# B&R Automation Studio project OpcUaSample410_BrbLibUa103 (part 7)

#### BrbUint64FromString.c
```c
#include <bur/plctypes.h>
#ifdef __cplusplus
	extern "C"
	{
#endif

#include "BrbLib.h"
#include <string.h>

#ifdef __cplusplus
	};
#endif

// NOLINTBEGIN(readability-*, bugprone-easily-swappable-parameters, clang-diagnostic-invalid-utf8, clang-diagnostic-invalid-source-encoding, clang-diagnostic-pointer-arith, clang-diagnostic-strict-prototypes, hicpp-uppercase-literal-suffix, cppcoreguidelines-*, performance-*)

// Die Matrix enthält für alle Dezimal-Wertigkeiten (0..9) jeder Stelle (0..19) die Bit-Wertigkeiten für Low+High
const BrbUint64_TYP BRBR_UINT64_FROMSTRING_MATRIX[20][10] =
	{
	//																0	Low      , High					1	Low      , High					2	Low      , High					3	Low      , High					4	Low      , High					5	Low      , High					6	Low      , High					7	Low      , High					8	Low      , High					9	Low      , High
	/* 00 = 1  */										{	{0x00000000, 0x00000000}, {0x00000001, 0x00000000}, {0x00000002, 0x00000000}, {0x00000003, 0x00000000}, {0x00000004, 0x00000000}, {0x00000005, 0x00000000}, {0x00000006, 0x00000000}, {0x00000007, 0x00000000}, {0x00000008, 0x00000000}, {0x00000009, 0x00000000}},
	/* 01 = 10 */										{	{0x00000000, 0x00000000}, {0x0000000A, 0x00000000}, {0x00000014, 0x00000000}, {0x0000001E, 0x00000000}, {0x00000028, 0x00000000}, {0x00000032, 0x00000000}, {0x0000003C, 0x00000000}, {0x00000046, 0x00000000}, {0x00000050, 0x00000000}, {0x0000005A, 0x00000000}},
	/* 02 = 100 */									{	{0x00000000, 0x00000000}, {0x00000064, 0x00000000}, {0x000000C8, 0x00000000}, {0x0000012C, 0x00000000}, {0x00000190, 0x00000000}, {0x000001F4, 0x00000000}, {0x00000258, 0x00000000}, {0x000002BC, 0x00000000}, {0x00000320, 0x00000000}, {0x00000384, 0x00000000}},
	/* 03 = 1000 */									{	{0x00000000, 0x00000000}, {0x000003E8, 0x00000000}, {0x000007D0, 0x00000000}, {0x00000BB8, 0x00000000}, {0x00000FA0, 0x00000000}, {0x00001388, 0x00000000}, {0x00001770, 0x00000000}, {0x00001B58, 0x00000000}, {0x00001F40, 0x00000000}, {0x00002328, 0x00000000}},
	/* 04 = 10000 */								{	{0x00000000, 0x00000000}, {0x00002710, 0x00000000}, {0x00004E20, 0x00000000}, {0x00007530, 0x00000000}, {0x00009C40, 0x00000000}, {0x0000C350, 0x00000000}, {0x0000EA60, 0x00000000}, {0x00011170, 0x00000000}, {0x00013880, 0x00000000}, {0x00015F90, 0x00000000}},
	/* 05 = 100000 */								{	{0x00000000, 0x00000000}, {0x000186A0, 0x00000000}, {0x00030D40, 0x00000000}, {0x000493E0, 0x00000000}, {0x00061A80, 0x00000000}, {0x0007A120, 0x00000000}, {0x000927C0, 0x00000000}, {0x000AAE60, 0x00000000}, {0x000C3500, 0x00000000}, {0x000DBBA0, 0x00000000}},
	/* 06 = 1000000 */							{	{0x00000000, 0x00000000}, {0x000F4240, 0x00000000}, {0x001E8480, 0x00000000}, {0x002DC6C0, 0x00000000}, {0x003D0900, 0x00000000}, {0x004C4B40, 0x00000000}, {0x005B8D80, 0x00000000}, {0x006ACFC0, 0x00000000}, {0x007A1200, 0x00000000}, {0x00895440, 0x00000000}},
	/* 07 = 10000000 */							{	{0x00000000, 0x00000000}, {0x00989680, 0x00000000}, {0x01312D00, 0x00000000}, {0x01C9C380, 0x00000000}, {0x02625A00, 0x00000000}, {0x02FAF080, 0x00000000}, {0x03938700, 0x00000000}, {0x042C1D80, 0x00000000}, {0x04C4B400, 0x00000000}, {0x055D4A80, 0x00000000}},
	/* 08 = 100000000 */						{	{0x00000000, 0x00000000}, {0x05F5E100, 0x00000000}, {0x0BEBC200, 0x00000000}, {0x11E1A300, 0x00000000}, {0x17D78400, 0x00000000}, {0x1DCD6500, 0x00000000}, {0x23C34600, 0x00000000}, {0x29B92700, 0x00000000}, {0x2FAF0800, 0x00000000}, {0x35A4E900, 0x00000000}},
	/* 09 = 1000000000 */						{	{0x00000000, 0x00000000}, {0x3B9ACA00, 0x00000000}, {0x77359400, 0x00000000}, {0xB2D05E00, 0x00000000}, {0xEE6B2800, 0x00000000}, {0x2A05F200, 0x00000001}, {0x65A0BC00, 0x00000001}, {0xA13B8600, 0x00000001}, {0xDCD65000, 0x00000001}, {0x18711A00, 0x00000002}},
	/* 10 = 10000000000 */					{	{0x00000000, 0x00000000}, {0x540BE400, 0x00000002}, {0xA817C800, 0x00000004}, {0xFC23AC00, 0x00000006}, {0x502F9000, 0x00000009}, {0xA43B7400, 0x0000000B}, {0xF8475800, 0x0000000D}, {0x4C533C00, 0x00000010}, {0xA05F2000, 0x00000012}, {0xF46B0400, 0x00000014}},
	/* 11 = 100000000000 */					{	{0x00000000, 0x00000000}, {0x4876E800, 0x00000017}, {0x90EDD000, 0x0000002E}, {0xD964B800, 0x00000045}, {0x21DBA000, 0x0000005D}, {0x6A528800, 0x00000074}, {0xB2C97000, 0x0000008B}, {0xFB405800, 0x000000A2}, {0x43B74000, 0x000000BA}, {0x8C2E2800, 0x000000D1}},
	/* 12 = 1000000000000 */				{	{0x00000000, 0x00000000}, {0xD4A51000, 0x000000E8}, {0xA94A2000, 0x000001D1}, {0x7DEF3000, 0x000002BA}, {0x52944000, 0x000003A3}, {0x27395000, 0x0000048C}, {0xFBDE6000, 0x00000574}, {0xD0837000, 0x0000065D}, {0xA5288000, 0x00000746}, {0x79CD9000, 0x0000082F}},
	/* 13 = 10000000000000 */				{	{0x00000000, 0x00000000}, {0x4E72A000, 0x00000918}, {0x9CE54000, 0x00001230}, {0xEB57E000, 0x00001B48}, {0x39CA8000, 0x00002461}, {0x883D2000, 0x00002D79}, {0xD6AFC000, 0x00003691}, {0x25226000, 0x00003FAA}, {0x73950000, 0x000048C2}, {0xC207A000, 0x000051DA}},
	/* 14 = 100000000000000 */			{	{0x00000000, 0x00000000}, {0x107A4000, 0x00005AF3}, {0x20F48000, 0x0000B5E6}, {0x316EC000, 0x000110D9}, {0x41E90000, 0x00016BCC}, {0x52634000, 0x0001C6BF}, {0x62DD8000, 0x000221B2}, {0x7357C000, 0x00027CA5}, {0x83D20000, 0x0002D798}, {0x944C4000, 0x0003328B}},
	/* 15 = 1000000000000000 */			{	{0x00000000, 0x00000000}, {0xA4C68000, 0x00038D7E}, {0x498D0000, 0x00071AFD}, {0xEE538000, 0x000AA87B}, {0x931A0000, 0x000E35FA}, {0x37E08000, 0x0011C379}, {0xDCA70000, 0x001550F7}, {0x816D8000, 0x0018DE76}, {0x26340000, 0x001C6BF5}, {0xCAFA8000, 0x001FF973}},
	/* 16 = 10000000000000000 */		{	{0x00000000, 0x00000000}, {0x6FC10000, 0x002386F2}, {0xDF820000, 0x00470DE4}, {0x4F430000, 0x006A94D7}, {0xBF040000, 0x008E1BC9}, {0x2EC50000, 0x00B1A2BC}, {0x9E860000, 0x00D529AE}, {0x0E470000, 0x00F8B0A1}, {0x7E080000, 0x011C3793}, {0xEDC90000, 0x013FBE85}},
	/* 17 = 100000000000000000 */		{	{0x00000000, 0x00000000}, {0x5D8A0000, 0x01634578}, {0xBB140000, 0x02C68AF0}, {0x189E0000, 0x0429D069}, {0x76280000, 0x058D15E1}, {0xD3B20000, 0x06F05B59}, {0x313C0000, 0x0853A0D2}, {0x8EC60000, 0x09B6E64A}, {0xEC500000, 0x0B1A2BC2}, {0x49DA0000, 0x0C7D713B}},
	/* 18 = 1000000000000000000 */	{	{0x00000000, 0x00000000}, {0xA7640000, 0x0DE0B6B3}, {0x4EC80000, 0x1BC16D67}, {0xF62C0000, 0x29A2241A}, {0x9D900000, 0x3782DACE}, {0x44F40000, 0x45639182}, {0xEC580000, 0x53444835}, {0x93BC0000, 0x6124FEE9}, {0x3B200000, 0x6F05B59D}, {0xE2840000, 0x7CE66C50}},
	/* 19 = 10000000000000000000 */	{	{0x00000000, 0x00000000}, {0x89E80000, 0x8AC72304}, {0x00000000, 0x00000000}, {0x00000000, 0x00000000}, {0x00000000, 0x00000000}, {0x00000000, 0x00000000}, {0x00000000, 0x00000000}, {0x00000000, 0x00000000}, {0x00000000, 0x00000000}, {0x00000000, 0x00000000}},
	};

/* Wandelt einen Uint64-Wert zu einem String */
signed long BrbUint64FromString(struct BrbUint64_TYP* pUint64, plcstring* pText)
{
	if(pUint64 == 0 || pText == 0)
	{
		return eBRB_ERR_NULL_POINTER;
	}
	pUint64->nLow = 0;
	pUint64->nHigh = 0;
	UDINT nTextLen = strlen(pText);
	if(nTextLen >= nBRB_UINT64_CHAR_MAX)
	{
		return eBRB_ERR_STRING_TOO_LONG;
	}
	DINT eResult = eBRB_ERR_OK;
	UDINT nDigit = 0; // Stelle von hinten
	STRING* pChar = 0;
	USINT nDigitVal = 0; // Wert der Stelle als Einer-Wertigkeit
	const BrbUint64_TYP* pOperand = 0; // Zeiger auf die Wertigkeits-Matrix
	for(nDigit=0; nDigit<nTextLen; nDigit++)
	{
		pChar = (STRING*)pText+(nTextLen-1-nDigit);
		if(*pChar >= '0' && *pChar <= '9')
		{
			// Zeichen ist eine Nummer
			nDigitVal = (USINT)(*pChar-'0'); // Wert als Einer-Stelle
			pOperand = &BRBR_UINT64_FROMSTRING_MATRIX[nDigit][nDigitVal];
			DINT nStatus = BrbByteArrayAdd((USINT*)pUint64, 8, (USINT*)pOperand, 8);
			if(nStatus != eBRB_ERR_OK)
			{
				// Überlauf -> Abbrechen
				eResult = nStatus;
				break;
			}
		}
		else
		{
			// Zeichen ist keine Nummer -> Abbrechen
			break;
		}
	}
	return eResult;
}

// NOLINTEND(readability-*, bugprone-easily-swappable-parameters, clang-diagnostic-invalid-utf8, clang-diagnostic-invalid-source-encoding, clang-diagnostic-pointer-arith, clang-diagnostic-strict-prototypes, hicpp-uppercase-literal-suffix, cppcoreguidelines-*, performance-*)
```

#### BrbUint64ToString.c
```c
#include <bur/plctypes.h>
#ifdef __cplusplus
	extern "C"
	{
#endif

#include "BrbLib.h"

#ifdef __cplusplus
	};
#endif

// NOLINTBEGIN(readability-*, bugprone-easily-swappable-parameters, clang-diagnostic-invalid-utf8, clang-diagnostic-invalid-source-encoding, clang-diagnostic-pointer-arith, clang-diagnostic-strict-prototypes, hicpp-uppercase-literal-suffix, cppcoreguidelines-*, performance-*)

typedef struct BrbUint64ToStringMatrixEntry_TYP
{
	unsigned long nBitMask;
	STRING sValueHigh[nBRB_UINT64_CHAR_MAX];
} BrbUint64ToStringMatrixEntry_TYP;

// Die Matrix enthält für alle Bit-Wertigkeiten (0..31) den IntegerString für High
const BrbUint64ToStringMatrixEntry_TYP BRBR_UINT64_TOSTRING_MATRIX[32] =
	{
	//							 nBitMask,	 sValueHigh
	/* Bit0  */			{0x00000001, "4294967296"},
	/* Bit1  */			{0x00000002, "8589934592"},
	/* Bit2  */			{0x00000004, "17179869184"},
	/* Bit3  */			{0x00000008, "34359738368"},
	/* Bit4  */			{0x00000010, "68719476736"},
	/* Bit5  */			{0x00000020, "137438953472"},
	/* Bit6  */			{0x00000040, "274877906944"},
	/* Bit7  */			{0x00000080, "549755813888"},
	/* Bit8  */			{0x00000100, "1099511627776"},
	/* Bit9  */			{0x00000200, "2199023255552"},
	/* Bit10 */			{0x00000400, "4398046511104"},
	/* Bit11 */			{0x00000800, "8796093022208"},
	/* Bit12 */			{0x00001000, "17592186044416"},
	/* Bit13 */			{0x00002000, "35184372088832"},
	/* Bit14 */			{0x00004000, "70368744177664"},
	/* Bit15 */			{0x00008000, "140737488355328"},
	/* Bit16 */			{0x00010000, "281474976710656"},
	/* Bit17 */			{0x00020000, "562949953421312"},
	/* Bit18 */			{0x00040000, "1125899906842624"},
	/* Bit19 */			{0x00080000, "2251799813685248"},
	/* Bit20 */			{0x00100000, "4503599627370496"},
	/* Bit21 */			{0x00200000, "9007199254740992"},
	/* Bit22 */			{0x00400000, "18014398509481984"},
	/* Bit23 */			{0x00800000, "36028797018963968"},
	/* Bit24 */			{0x01000000, "72057594037927936"},
	/* Bit25 */			{0x02000000, "144115188075855872"},
	/* Bit26 */			{0x04000000, "288230376151711744"},
	/* Bit27 */			{0x08000000, "576460752303423488"},
	/* Bit28 */			{0x10000000, "1152921504606846976"},
	/* Bit29 */			{0x20000000, "2305843009213693952"},
	/* Bit30 */			{0x40000000, "4611686018427387904"},
	/* Bit31 */			{0x80000000, "9223372036854775808"},
	};

/* Wandelt einen Uint64-Wert zu einem String */
signed long BrbUint64ToString(struct BrbUint64_TYP* pUint64, plcstring* pText, unsigned long nTextSize)
{
	if(pUint64 == 0 || pText == 0)
	{
		return eBRB_ERR_NULL_POINTER;
	}
	if(nTextSize < nBRB_UINT64_CHAR_MAX)
	{
		return eBRB_ERR_STRING_TOO_SHORT;
	}
	// Wandlung Low
	BrbUdintToAscii(pUint64->nLow, pText);
	// Wandlung High
	// Der C-Befehl sprintf ist leider auf der Sps nicht erlaubt. Daher wird für jedes der 32 Bits die Wertigkeit addiert.
	USINT nBit = 0;
	for(nBit=0; nBit<=31; nBit++)
	{
		const BrbUint64ToStringMatrixEntry_TYP* pMatrixEntry = &BRBR_UINT64_TOSTRING_MATRIX[nBit];
		if(pUint64->nHigh & pMatrixEntry->nBitMask)
		{
			BrbIntegerStringAdd(pText, (STRING*)&pMatrixEntry->sValueHigh, nBRB_UINT64_CHAR_MAX);
		}
	}
	return eBRB_ERR_OK;
}

// NOLINTEND(readability-*, bugprone-easily-swappable-parameters, clang-diagnostic-invalid-utf8, clang-diagnostic-invalid-source-encoding, clang-diagnostic-pointer-arith, clang-diagnostic-strict-prototypes, hicpp-uppercase-literal-suffix, cppcoreguidelines-*, performance-*)
```

#### BrbUint64Compare.c
```c
#include <bur/plctypes.h>
#ifdef __cplusplus
	extern "C"
	{
#endif

#include "BrbLib.h"

#ifdef __cplusplus
	};
#endif

// NOLINTBEGIN(readability-*, bugprone-easily-swappable-parameters, clang-diagnostic-invalid-utf8, clang-diagnostic-invalid-source-encoding, clang-diagnostic-pointer-arith, clang-diagnostic-strict-prototypes, hicpp-uppercase-literal-suffix, cppcoreguidelines-*, performance-*)

/* Vergleicht zwei Uint64 auf kleiner, größer oder gleich */
signed char BrbUint64Compare(struct BrbUint64_TYP* pOperand0, struct BrbUint64_TYP* pOperand1)
{
	if(pOperand0 == 0 || pOperand1 == 0)
	{
		return 0;
	}
	SINT nResult = 0;
	// NOLINTBEGIN(bugprone-branch-clone)
	if(pOperand0->nHigh > pOperand1->nHigh)
	{
		nResult = 1;
	}
	else if(pOperand0->nHigh < pOperand1->nHigh)
	{
		nResult = -1;
	}
	else if(pOperand0->nLow > pOperand1->nLow)
	{
		nResult = 1;
	}
	else if(pOperand0->nLow < pOperand1->nLow)
	{
		nResult = -1;
	}
	// NOLINTEND(bugprone-branch-clone)
	return nResult;
}

// NOLINTEND(readability-*, bugprone-easily-swappable-parameters, clang-diagnostic-invalid-utf8, clang-diagnostic-invalid-source-encoding, clang-diagnostic-pointer-arith, clang-diagnostic-strict-prototypes, hicpp-uppercase-literal-suffix, cppcoreguidelines-*, performance-*)
```

#### BrbUint64Inc.c
```c
#include <bur/plctypes.h>
#ifdef __cplusplus
	extern "C"
	{
#endif

#include "BrbLib.h"

#ifdef __cplusplus
	};
#endif

// NOLINTBEGIN(readability-*, bugprone-easily-swappable-parameters, clang-diagnostic-invalid-utf8, clang-diagnostic-invalid-source-encoding, clang-diagnostic-pointer-arith, clang-diagnostic-strict-prototypes, hicpp-uppercase-literal-suffix, cppcoreguidelines-*, performance-*)

/* Inkrementiert einen Uint64-Wert um 1 */
signed long BrbUint64Inc(struct BrbUint64_TYP* pUint64)
{
	if(pUint64 == 0)
	{
		return eBRB_ERR_NULL_POINTER;
	}
	BrbUint64_TYP nOperand;
	nOperand.nLow = 1;
	nOperand.nHigh = 0;
	return BrbUint64Calculate(pUint64, &nOperand, eBRB_DT64_OPERATOR_ADD);
}

// NOLINTEND(readability-*, bugprone-easily-swappable-parameters, clang-diagnostic-invalid-utf8, clang-diagnostic-invalid-source-encoding, clang-diagnostic-pointer-arith, clang-diagnostic-strict-prototypes, hicpp-uppercase-literal-suffix, cppcoreguidelines-*, performance-*)
```

#### BrbUint64Dec.c
```c
#include <bur/plctypes.h>
#ifdef __cplusplus
	extern "C"
	{
#endif

#include "BrbLib.h"

#ifdef __cplusplus
	};
#endif

// NOLINTBEGIN(readability-*, bugprone-easily-swappable-parameters, clang-diagnostic-invalid-utf8, clang-diagnostic-invalid-source-encoding, clang-diagnostic-pointer-arith, clang-diagnostic-strict-prototypes, hicpp-uppercase-literal-suffix, cppcoreguidelines-*, performance-*)

/* Dekrementiert einen Uint64-Wert um 1 */
signed long BrbUint64Dec(struct BrbUint64_TYP* pUint64)
{
	if(pUint64 == 0)
	{
		return eBRB_ERR_NULL_POINTER;
	}
	BrbUint64_TYP nOperand;
	nOperand.nLow = 1;
	nOperand.nHigh = 0;
	return BrbUint64Calculate(pUint64, &nOperand, eBRB_DT64_OPERATOR_SUBTRACT);
}

// NOLINTEND(readability-*, bugprone-easily-swappable-parameters, clang-diagnostic-invalid-utf8, clang-diagnostic-invalid-source-encoding, clang-diagnostic-pointer-arith, clang-diagnostic-strict-prototypes, hicpp-uppercase-literal-suffix, cppcoreguidelines-*, performance-*)
```

#### BrbUint64Calculate.c
```c
#include <bur/plctypes.h>
#ifdef __cplusplus
	extern "C"
	{
#endif

#include "BrbLib.h"

#ifdef __cplusplus
	};
#endif

// NOLINTBEGIN(readability-*, bugprone-easily-swappable-parameters, clang-diagnostic-invalid-utf8, clang-diagnostic-invalid-source-encoding, clang-diagnostic-pointer-arith, clang-diagnostic-strict-prototypes, hicpp-uppercase-literal-suffix, cppcoreguidelines-*, performance-*)

/* Rechnet mit zwei Uint64 */
signed long BrbUint64Calculate(struct BrbUint64_TYP* pOperand0, struct BrbUint64_TYP* pOperand1, enum BrbDt64Operator_ENUM eOperator)
{
	if(pOperand0 == 0 || pOperand1 == 0)
	{
		return eBRB_ERR_NULL_POINTER;
	}
	unsigned long long* pUlintOperand0 = (unsigned long long*)pOperand0;
	unsigned long long* pUlintOperand1 = (unsigned long long*)pOperand1;
	switch(eOperator) // NOLINT(hicpp-multiway-paths-covered)
	{
		case eBRB_DT64_OPERATOR_ADD:
			*pUlintOperand0 = *pUlintOperand0 + *pUlintOperand1;
			break;

		case eBRB_DT64_OPERATOR_SUBTRACT:
			*pUlintOperand0 = *pUlintOperand0 - *pUlintOperand1;
			break;

		case eBRB_DT64_OPERATOR_MULTIPLY:
			*pUlintOperand0 = *pUlintOperand0 * *pUlintOperand1;
			break;

		case eBRB_DT64_OPERATOR_DIVIDE:
			if(*pUlintOperand1 == 0)
			{
				return eBRB_ERR_DIVISION_BY_0;
			}
			*pUlintOperand0 = *pUlintOperand0 / *pUlintOperand1;
			break;

	}
	return eBRB_ERR_OK;
}

// NOLINTEND(readability-*, bugprone-easily-swappable-parameters, clang-diagnostic-invalid-utf8, clang-diagnostic-invalid-source-encoding, clang-diagnostic-pointer-arith, clang-diagnostic-strict-prototypes, hicpp-uppercase-literal-suffix, cppcoreguidelines-*, performance-*)
```

#### BrbInt64FromString.c
```c
#include <bur/plctypes.h>
#ifdef __cplusplus
	extern "C"
	{
#endif

#include "BrbLib.h"
#include <string.h>

#ifdef __cplusplus
	};
#endif

// NOLINTBEGIN(readability-*, bugprone-easily-swappable-parameters, clang-diagnostic-invalid-utf8, clang-diagnostic-invalid-source-encoding, clang-diagnostic-pointer-arith, clang-diagnostic-strict-prototypes, hicpp-uppercase-literal-suffix, cppcoreguidelines-*, performance-*)

// Die Matrix enthält für alle Dezimal-Wertigkeiten (0..9) jeder Stelle (0..19) die Bit-Wertigkeiten für Low+High
const BrbInt64_TYP nBRB_INT64_VALENCY_MATRIX[19][10] =
	{
	//																0	Low      , High					1	Low      , High					2	Low      , High					3	Low      , High					4	Low      , High					5	Low      , High					6	Low      , High					7	Low      , High					8	Low      , High					9	Low      , High
	/* 00 = 1  */										{	{0x00000000, 0x00000000}, {0x00000001, 0x00000000}, {0x00000002, 0x00000000}, {0x00000003, 0x00000000}, {0x00000004, 0x00000000}, {0x00000005, 0x00000000}, {0x00000006, 0x00000000}, {0x00000007, 0x00000000}, {0x00000008, 0x00000000}, {0x00000009, 0x00000000}},
	/* 01 = 10 */										{	{0x00000000, 0x00000000}, {0x0000000A, 0x00000000}, {0x00000014, 0x00000000}, {0x0000001E, 0x00000000}, {0x00000028, 0x00000000}, {0x00000032, 0x00000000}, {0x0000003C, 0x00000000}, {0x00000046, 0x00000000}, {0x00000050, 0x00000000}, {0x0000005A, 0x00000000}},
	/* 02 = 100 */									{	{0x00000000, 0x00000000}, {0x00000064, 0x00000000}, {0x000000C8, 0x00000000}, {0x0000012C, 0x00000000}, {0x00000190, 0x00000000}, {0x000001F4, 0x00000000}, {0x00000258, 0x00000000}, {0x000002BC, 0x00000000}, {0x00000320, 0x00000000}, {0x00000384, 0x00000000}},
	/* 03 = 1000 */									{	{0x00000000, 0x00000000}, {0x000003E8, 0x00000000}, {0x000007D0, 0x00000000}, {0x00000BB8, 0x00000000}, {0x00000FA0, 0x00000000}, {0x00001388, 0x00000000}, {0x00001770, 0x00000000}, {0x00001B58, 0x00000000}, {0x00001F40, 0x00000000}, {0x00002328, 0x00000000}},
	/* 04 = 10000 */								{	{0x00000000, 0x00000000}, {0x00002710, 0x00000000}, {0x00004E20, 0x00000000}, {0x00007530, 0x00000000}, {0x00009C40, 0x00000000}, {0x0000C350, 0x00000000}, {0x0000EA60, 0x00000000}, {0x00011170, 0x00000000}, {0x00013880, 0x00000000}, {0x00015F90, 0x00000000}},
	/* 05 = 100000 */								{	{0x00000000, 0x00000000}, {0x000186A0, 0x00000000}, {0x00030D40, 0x00000000}, {0x000493E0, 0x00000000}, {0x00061A80, 0x00000000}, {0x0007A120, 0x00000000}, {0x000927C0, 0x00000000}, {0x000AAE60, 0x00000000}, {0x000C3500, 0x00000000}, {0x000DBBA0, 0x00000000}},
	/* 06 = 1000000 */							{	{0x00000000, 0x00000000}, {0x000F4240, 0x00000000}, {0x001E8480, 0x00000000}, {0x002DC6C0, 0x00000000}, {0x003D0900, 0x00000000}, {0x004C4B40, 0x00000000}, {0x005B8D80, 0x00000000}, {0x006ACFC0, 0x00000000}, {0x007A1200, 0x00000000}, {0x00895440, 0x00000000}},
	/* 07 = 10000000 */							{	{0x00000000, 0x00000000}, {0x00989680, 0x00000000}, {0x01312D00, 0x00000000}, {0x01C9C380, 0x00000000}, {0x02625A00, 0x00000000}, {0x02FAF080, 0x00000000}, {0x03938700, 0x00000000}, {0x042C1D80, 0x00000000}, {0x04C4B400, 0x00000000}, {0x055D4A80, 0x00000000}},
	/* 08 = 100000000 */						{	{0x00000000, 0x00000000}, {0x05F5E100, 0x00000000}, {0x0BEBC200, 0x00000000}, {0x11E1A300, 0x00000000}, {0x17D78400, 0x00000000}, {0x1DCD6500, 0x00000000}, {0x23C34600, 0x00000000}, {0x29B92700, 0x00000000}, {0x2FAF0800, 0x00000000}, {0x35A4E900, 0x00000000}},
	/* 09 = 1000000000 */						{	{0x00000000, 0x00000000}, {0x3B9ACA00, 0x00000000}, {0x77359400, 0x00000000}, {0xB2D05E00, 0x00000000}, {0xEE6B2800, 0x00000000}, {0x2A05F200, 0x00000001}, {0x65A0BC00, 0x00000001}, {0xA13B8600, 0x00000001}, {0xDCD65000, 0x00000001}, {0x18711A00, 0x00000002}},
	/* 10 = 10000000000 */					{	{0x00000000, 0x00000000}, {0x540BE400, 0x00000002}, {0xA817C800, 0x00000004}, {0xFC23AC00, 0x00000006}, {0x502F9000, 0x00000009}, {0xA43B7400, 0x0000000B}, {0xF8475800, 0x0000000D}, {0x4C533C00, 0x00000010}, {0xA05F2000, 0x00000012}, {0xF46B0400, 0x00000014}},
	/* 11 = 100000000000 */					{	{0x00000000, 0x00000000}, {0x4876E800, 0x00000017}, {0x90EDD000, 0x0000002E}, {0xD964B800, 0x00000045}, {0x21DBA000, 0x0000005D}, {0x6A528800, 0x00000074}, {0xB2C97000, 0x0000008B}, {0xFB405800, 0x000000A2}, {0x43B74000, 0x000000BA}, {0x8C2E2800, 0x000000D1}},
	/* 12 = 1000000000000 */				{	{0x00000000, 0x00000000}, {0xD4A51000, 0x000000E8}, {0xA94A2000, 0x000001D1}, {0x7DEF3000, 0x000002BA}, {0x52944000, 0x000003A3}, {0x27395000, 0x0000048C}, {0xFBDE6000, 0x00000574}, {0xD0837000, 0x0000065D}, {0xA5288000, 0x00000746}, {0x79CD9000, 0x0000082F}},
	/* 13 = 10000000000000 */				{	{0x00000000, 0x00000000}, {0x4E72A000, 0x00000918}, {0x9CE54000, 0x00001230}, {0xEB57E000, 0x00001B48}, {0x39CA8000, 0x00002461}, {0x883D2000, 0x00002D79}, {0xD6AFC000, 0x00003691}, {0x25226000, 0x00003FAA}, {0x73950000, 0x000048C2}, {0xC207A000, 0x000051DA}},
	/* 14 = 100000000000000 */			{	{0x00000000, 0x00000000}, {0x107A4000, 0x00005AF3}, {0x20F48000, 0x0000B5E6}, {0x316EC000, 0x000110D9}, {0x41E90000, 0x00016BCC}, {0x52634000, 0x0001C6BF}, {0x62DD8000, 0x000221B2}, {0x7357C000, 0x00027CA5}, {0x83D20000, 0x0002D798}, {0x944C4000, 0x0003328B}},
	/* 15 = 1000000000000000 */			{	{0x00000000, 0x00000000}, {0xA4C68000, 0x00038D7E}, {0x498D0000, 0x00071AFD}, {0xEE538000, 0x000AA87B}, {0x931A0000, 0x000E35FA}, {0x37E08000, 0x0011C379}, {0xDCA70000, 0x001550F7}, {0x816D8000, 0x0018DE76}, {0x26340000, 0x001C6BF5}, {0xCAFA8000, 0x001FF973}},
	/* 16 = 10000000000000000 */		{	{0x00000000, 0x00000000}, {0x6FC10000, 0x002386F2}, {0xDF820000, 0x00470DE4}, {0x4F430000, 0x006A94D7}, {0xBF040000, 0x008E1BC9}, {0x2EC50000, 0x00B1A2BC}, {0x9E860000, 0x00D529AE}, {0x0E470000, 0x00F8B0A1}, {0x7E080000, 0x011C3793}, {0xEDC90000, 0x013FBE85}},
	/* 17 = 100000000000000000 */		{	{0x00000000, 0x00000000}, {0x5D8A0000, 0x01634578}, {0xBB140000, 0x02C68AF0}, {0x189E0000, 0x0429D069}, {0x76280000, 0x058D15E1}, {0xD3B20000, 0x06F05B59}, {0x313C0000, 0x0853A0D2}, {0x8EC60000, 0x09B6E64A}, {0xEC500000, 0x0B1A2BC2}, {0x49DA0000, 0x0C7D713B}},
	/* 18 = 1000000000000000000 */	{	{0x00000000, 0x00000000}, {0xA7640000, 0x0DE0B6B3}, {0x4EC80000, 0x1BC16D67}, {0xF62C0000, 0x29A2241A}, {0x9D900000, 0x3782DACE}, {0x44F40000, 0x45639182}, {0xEC580000, 0x53444835}, {0x93BC0000, 0x6124FEE9}, {0x3B200000, 0x6F05B59D}, {0xE2840000, 0x7CE66C50}},
	};

/* Wandelt einen Int64-Wert zu einem String */
signed long BrbInt64FromString(struct BrbInt64_TYP* pInt64, plcstring* pText) // NOLINT(readability-function-cognitive-complexity)
{
	if(pInt64 == 0 || pText == 0)
	{
		return eBRB_ERR_NULL_POINTER;
	}
	UDINT nTextLen = strlen(pText);
	if(BrbStringStartsWith(pText, "-") == 1)
	{
		// Negative Zahl
		if(nTextLen >= nBRB_INT64_CHAR_MAX)
		{
			return eBRB_ERR_STRING_TOO_LONG;
		}
		pInt64->nLow = 0;
		pInt64->nHigh = 0;
		UDINT nDigit = 0; // Stelle von hinten
		STRING* pChar = 0;
		USINT nDigitVal = 0; // Wert der Stelle als Einer-Wertigkeit
		const BrbInt64_TYP* pOperand = 0; // Zeiger auf die Wertigkeits-Matrix
		for(nDigit=0; nDigit<nTextLen; nDigit++)
		{
			pChar = (STRING*)pText+(nTextLen-1-nDigit);
			if(*pChar >= '0' && *pChar <= '9')
			{
				// Zeichen ist eine Nummer
				nDigitVal = (USINT)(*pChar-'0'); // Wert als Einer-Stelle
				pOperand = &nBRB_INT64_VALENCY_MATRIX[nDigit][nDigitVal];
				BrbByteArraySubtract((USINT*)pInt64, 8, (USINT*)pOperand, 8);
			}
			else
			{
				// Zeichen ist keine Nummer -> Abbrechen
				break;
			}
		}
		if((pInt64->nHigh & 0x80000000) == 0)
		{
			// Unterlauf
			return eBRB_ERR_OVERFLOW;
		}
	}
	else
	{
		// Postive Zahl
		if(nTextLen >= nBRB_INT64_CHAR_MAX-1)
		{
			return eBRB_ERR_STRING_TOO_LONG;
		}
		pInt64->nLow = 0;
		pInt64->nHigh = 0;
		UDINT nDigit = 0; // Stelle von hinten
		STRING* pChar = 0;
		USINT nDigitVal = 0; // Wert der Stelle als Einer-Wertigkeit
		const BrbInt64_TYP* pOperand = 0; // Zeiger auf die Wertigkeits-Matrix
		for(nDigit=0; nDigit<nTextLen; nDigit++)
		{
			pChar = (STRING*)pText+(nTextLen-1-nDigit);
			if(*pChar >= '0' && *pChar <= '9')
			{
				// Zeichen ist eine Nummer
				nDigitVal = (USINT)(*pChar-'0'); // Wert als Einer-Stelle
				pOperand = &nBRB_INT64_VALENCY_MATRIX[nDigit][nDigitVal];
				BrbByteArrayAdd((USINT*)pInt64, 8, (USINT*)pOperand, 8);
				if((pInt64->nHigh & 0x80000000) > 0)
				{
					// Überlauf -> Abbrechen
					return eBRB_ERR_OVERFLOW;
				}
			}
			else
			{
				// Zeichen ist keine Nummer -> Abbrechen
				break;
			}
		}
	}
	return eBRB_ERR_OK;
}

// NOLINTEND(readability-*, bugprone-easily-swappable-parameters, clang-diagnostic-invalid-utf8, clang-diagnostic-invalid-source-encoding, clang-diagnostic-pointer-arith, clang-diagnostic-strict-prototypes, hicpp-uppercase-literal-suffix, cppcoreguidelines-*, performance-*)
```

#### BrbInt64ToString.c
```c
#include <bur/plctypes.h>
#ifdef __cplusplus
	extern "C"
	{
#endif

#include "BrbLib.h"

#ifdef __cplusplus
	};
#endif

// NOLINTBEGIN(readability-*, bugprone-easily-swappable-parameters, clang-diagnostic-invalid-utf8, clang-diagnostic-invalid-source-encoding, clang-diagnostic-pointer-arith, clang-diagnostic-strict-prototypes, hicpp-uppercase-literal-suffix, cppcoreguidelines-*, performance-*)

typedef struct BrbUint64ToStringMatrixEntry_TYP
{
	unsigned long nBitMask;
	STRING sValueLow[nBRB_INT64_CHAR_MAX];
	STRING sValueHigh[nBRB_INT64_CHAR_MAX];
} BrbInt64ToStringMatrixEntry_TYP;

// Die Matrix enthält für alle Bit-Wertigkeiten (0..31) den IntegerString für Low und High
const BrbInt64ToStringMatrixEntry_TYP BRBR_INT64_TOSTRING_MATRIX[32] =
	{
	//							 nBitMask,	 sValueLow,			sValueHigh
	/* Bit0  */			{0x00000001, "1",						"4294967296"},
	/* Bit1  */			{0x00000002, "2",						"8589934592"},
	/* Bit2  */			{0x00000004, "4",						"17179869184"},
	/* Bit3  */			{0x00000008, "8",						"34359738368"},
	/* Bit4  */			{0x00000010, "16",					"68719476736"},
	/* Bit5  */			{0x00000020, "32",					"137438953472"},
	/* Bit6  */			{0x00000040, "64",					"274877906944"},
	/* Bit7  */			{0x00000080, "128",					"549755813888"},
	/* Bit8  */			{0x00000100, "256",					"1099511627776"},
	/* Bit9  */			{0x00000200, "512",					"2199023255552"},
	/* Bit10 */			{0x00000400, "1024",				"4398046511104"},
	/* Bit11 */			{0x00000800, "2048",				"8796093022208"},
	/* Bit12 */			{0x00001000, "4096",				"17592186044416"},
	/* Bit13 */			{0x00002000, "8192",				"35184372088832"},
	/* Bit14 */			{0x00004000, "16384",				"70368744177664"},
	/* Bit15 */			{0x00008000, "32768",				"140737488355328"},
	/* Bit16 */			{0x00010000, "65536",				"281474976710656"},
	/* Bit17 */			{0x00020000, "131072",			"562949953421312"},
	/* Bit18 */			{0x00040000, "262144",			"1125899906842624"},
	/* Bit19 */			{0x00080000, "524288",			"2251799813685248"},
	/* Bit20 */			{0x00100000, "1048576",			"4503599627370496"},
	/* Bit21 */			{0x00200000, "2097152",			"9007199254740992"},
	/* Bit22 */			{0x00400000, "4194304",			"18014398509481984"},
	/* Bit23 */			{0x00800000, "8388608",			"36028797018963968"},
	/* Bit24 */			{0x01000000, "16777216",		"72057594037927936"},
	/* Bit25 */			{0x02000000, "33554432",		"144115188075855872"},
	/* Bit26 */			{0x04000000, "67108864",		"288230376151711744"},
	/* Bit27 */			{0x08000000, "134217728",		"576460752303423488"},
	/* Bit28 */			{0x10000000, "268435456",		"1152921504606846976"},
	/* Bit29 */			{0x20000000, "536870912",		"2305843009213693952"},
	/* Bit30 */			{0x40000000, "1073741824",	"4611686018427387904"},
	/* Bit31 */			{0x80000000, "2147483648",	"0"}
	};

/* Wandelt einen Int64-Wert zu einem String */
signed long BrbInt64ToString(struct BrbInt64_TYP* pInt64, plcstring* pText, unsigned long nTextSize) // NOLINT(readability-function-cognitive-complexity)
{
	if(pInt64 == 0 || pText == 0)
	{
		return eBRB_ERR_NULL_POINTER;
	}
	if(nTextSize < nBRB_INT64_CHAR_MAX)
	{
		return eBRB_ERR_STRING_TOO_SHORT;
	}
	// Der C-Befehl sprintf ist leider auf der Sps nicht erlaubt.  Daher wird für jedes der 31 Bits die Wertigkeit addiert.
	if((pInt64->nHigh & 0x80000000) == 0)
	{
		// Positiv
		// Wandlung Low
		BrbUdintToAscii(pInt64->nLow, pText);
		// Wandlung High
		USINT nBit = 0;
		for(nBit=0; nBit<=30; nBit++)
		{
			const BrbInt64ToStringMatrixEntry_TYP* pMatrixEntry = &BRBR_INT64_TOSTRING_MATRIX[nBit];
			if(pInt64->nHigh & pMatrixEntry->nBitMask)
			{
				BrbIntegerStringAdd(pText, (STRING*)&pMatrixEntry->sValueHigh, nBRB_INT64_CHAR_MAX);
			}
		}
	}
	else
	{
		// Negativ
		// Wandlung Low
		BrbStringCopy(pText, "0", nBRB_INT64_CHAR_MAX+1);
		BrbIntegerStringAdd(pText, "1", nBRB_INT64_CHAR_MAX+1);
		USINT nBit = 0;
		for(nBit=0; nBit<=31; nBit++)
		{
			const BrbInt64ToStringMatrixEntry_TYP* pMatrixEntry = &BRBR_INT64_TOSTRING_MATRIX[nBit];
			if((pInt64->nLow & pMatrixEntry->nBitMask) == 0)
			{
				BrbIntegerStringAdd(pText, (STRING*)&pMatrixEntry->sValueLow, nBRB_INT64_CHAR_MAX);
			}
		}
		// Wandlung High
		for(nBit=0; nBit<=30; nBit++)
		{
			const BrbInt64ToStringMatrixEntry_TYP* pMatrixEntry = &BRBR_INT64_TOSTRING_MATRIX[nBit];
			if((pInt64->nHigh & pMatrixEntry->nBitMask) == 0)
			{
				BrbIntegerStringAdd(pText, (STRING*)&pMatrixEntry->sValueHigh, nBRB_INT64_CHAR_MAX);
			}
		}
		// Minuszeichen
		BrbStringInsert(pText, 0, "-");
	}
	return eBRB_ERR_OK;
}

// NOLINTEND(readability-*, bugprone-easily-swappable-parameters, clang-diagnostic-invalid-utf8, clang-diagnostic-invalid-source-encoding, clang-diagnostic-pointer-arith, clang-diagnostic-strict-prototypes, hicpp-uppercase-literal-suffix, cppcoreguidelines-*, performance-*)
```

#### BrbInt64Compare.c
```c
#include <bur/plctypes.h>
#ifdef __cplusplus
	extern "C"
	{
#endif

#include "BrbLib.h"

#ifdef __cplusplus
	};
#endif

// NOLINTBEGIN(readability-*, bugprone-easily-swappable-parameters, clang-diagnostic-invalid-utf8, clang-diagnostic-invalid-source-encoding, clang-diagnostic-pointer-arith, clang-diagnostic-strict-prototypes, hicpp-uppercase-literal-suffix, cppcoreguidelines-*, performance-*)

/* Vergleicht zwei Int64 auf kleiner, größer oder gleich */
signed char BrbInt64Compare(struct BrbInt64_TYP* pOperand0, struct BrbInt64_TYP* pOperand1)
{
	if(pOperand0 == 0 || pOperand1 == 0)
	{
		return 0;
	}
	SINT nResult = 0;
	BOOL bNegativeBit0 = (pOperand0->nHigh & 0x80000000) == 0x80000000;
	BOOL bNegativeBit1 = (pOperand1->nHigh & 0x80000000) == 0x80000000;
	if(bNegativeBit0 == 0 && bNegativeBit1 == 1)
	{
		// 0=Positiv, 1=Negativ
		nResult = 1;
	}
	else if(bNegativeBit0 == 1 && bNegativeBit1 == 0)
	{
		// 0=Negativ, 1=Positiv
		nResult = -1;
	}
	else
	{
		// Beide positiv oder beide negativ
		UDINT nHigh0 = pOperand0->nHigh & 0x7FFFFFFF; // NOLINT(hicpp-signed-bitwise)
		UDINT nHigh1 = pOperand1->nHigh & 0x7FFFFFFF; // NOLINT(hicpp-signed-bitwise)
		// NOLINTBEGIN(bugprone-branch-clone)
		if(nHigh0 > nHigh1)
		{
			nResult = 1;
		}
		else if(nHigh0 < nHigh1)
		{
			nResult = -1;
		}
		else if(pOperand0->nLow > pOperand1->nLow)
		{
			nResult = 1;
		}
		else if(pOperand0->nLow < pOperand1->nLow)
		{
			nResult = -1;
		}
		// NOLINTEND(bugprone-branch-clone)
	}
	return nResult;
}

// NOLINTEND(readability-*, bugprone-easily-swappable-parameters, clang-diagnostic-invalid-utf8, clang-diagnostic-invalid-source-encoding, clang-diagnostic-pointer-arith, clang-diagnostic-strict-prototypes, hicpp-uppercase-literal-suffix, cppcoreguidelines-*, performance-*)
```

#### BrbInt64Inc.c
```c
#include <bur/plctypes.h>
#ifdef __cplusplus
	extern "C"
	{
#endif

#include "BrbLib.h"

#ifdef __cplusplus
	};
#endif

// NOLINTBEGIN(readability-*, bugprone-easily-swappable-parameters, clang-diagnostic-invalid-utf8, clang-diagnostic-invalid-source-encoding, clang-diagnostic-pointer-arith, clang-diagnostic-strict-prototypes, hicpp-uppercase-literal-suffix, cppcoreguidelines-*, performance-*)

/* Inkrementiert einen Int64-Wert um 1 */
signed long BrbInt64Inc(struct BrbInt64_TYP* pInt64)
{
	if(pInt64 == 0)
	{
		return eBRB_ERR_NULL_POINTER;
	}
	BrbInt64_TYP nOperand;
	nOperand.nLow = 1;
	nOperand.nHigh = 0;
	return BrbInt64Calculate(pInt64, &nOperand, eBRB_DT64_OPERATOR_ADD);
}

// NOLINTEND(readability-*, bugprone-easily-swappable-parameters, clang-diagnostic-invalid-utf8, clang-diagnostic-invalid-source-encoding, clang-diagnostic-pointer-arith, clang-diagnostic-strict-prototypes, hicpp-uppercase-literal-suffix, cppcoreguidelines-*, performance-*)
```

#### BrbInt64Dec.c
```c
#include <bur/plctypes.h>
#ifdef __cplusplus
	extern "C"
	{
#endif

#include "BrbLib.h"

#ifdef __cplusplus
	};
#endif

// NOLINTBEGIN(readability-*, bugprone-easily-swappable-parameters, clang-diagnostic-invalid-utf8, clang-diagnostic-invalid-source-encoding, clang-diagnostic-pointer-arith, clang-diagnostic-strict-prototypes, hicpp-uppercase-literal-suffix, cppcoreguidelines-*, performance-*)

/* Dekrementiert einen Int64-Wert um 1 */
signed long BrbInt64Dec(struct BrbInt64_TYP* pInt64)
{
	if(pInt64 == 0)
	{
		return eBRB_ERR_NULL_POINTER;
	}
	BrbInt64_TYP nOperand;
	nOperand.nLow = 1;
	nOperand.nHigh = 0;
	return BrbInt64Calculate(pInt64, &nOperand, eBRB_DT64_OPERATOR_SUBTRACT);
}

// NOLINTEND(readability-*, bugprone-easily-swappable-parameters, clang-diagnostic-invalid-utf8, clang-diagnostic-invalid-source-encoding, clang-diagnostic-pointer-arith, clang-diagnostic-strict-prototypes, hicpp-uppercase-literal-suffix, cppcoreguidelines-*, performance-*)
```

#### BrbInt64Calculate.c
```c
#include <bur/plctypes.h>
#ifdef __cplusplus
	extern "C"
	{
#endif

#include "BrbLib.h"

#ifdef __cplusplus
	};
#endif

// NOLINTBEGIN(readability-*, bugprone-easily-swappable-parameters, clang-diagnostic-invalid-utf8, clang-diagnostic-invalid-source-encoding, clang-diagnostic-pointer-arith, clang-diagnostic-strict-prototypes, hicpp-uppercase-literal-suffix, cppcoreguidelines-*, performance-*)

/* Rechnet mit zwei Int64 */
signed long BrbInt64Calculate(struct BrbInt64_TYP* pOperand0, struct BrbInt64_TYP* pOperand1, enum BrbDt64Operator_ENUM eOperator)
{
	if(pOperand0 == 0 || pOperand1 == 0)
	{
		return eBRB_ERR_NULL_POINTER;
	}
	signed long long* pLintOperand0 = (signed long long*)pOperand0;
	signed long long* pLintOperand1 = (signed long long*)pOperand1;
	switch(eOperator) // NOLINT(hicpp-multiway-paths-covered)
	{
		case eBRB_DT64_OPERATOR_ADD:
			*pLintOperand0 = *pLintOperand0 + *pLintOperand1;
			break;

		case eBRB_DT64_OPERATOR_SUBTRACT:
			*pLintOperand0 = *pLintOperand0 - *pLintOperand1;
			break;

		case eBRB_DT64_OPERATOR_MULTIPLY:
			*pLintOperand0 = *pLintOperand0 * *pLintOperand1;
			break;

		case eBRB_DT64_OPERATOR_DIVIDE:
			if(*pLintOperand1 == 0)
			{
				return eBRB_ERR_DIVISION_BY_0;
			}
			*pLintOperand0 = *pLintOperand0 / *pLintOperand1;
			break;

	}
	return eBRB_ERR_OK;
}

// NOLINTEND(readability-*, bugprone-easily-swappable-parameters, clang-diagnostic-invalid-utf8, clang-diagnostic-invalid-source-encoding, clang-diagnostic-pointer-arith, clang-diagnostic-strict-prototypes, hicpp-uppercase-literal-suffix, cppcoreguidelines-*, performance-*)
```

#### BrbIntegerStringAdd.c
```c
#include <bur/plctypes.h>
#ifdef __cplusplus
	extern "C"
	{
#endif

#include "BrbLib.h"
#include <string.h>

#ifdef __cplusplus
	};
#endif

// NOLINTBEGIN(readability-*, bugprone-easily-swappable-parameters, clang-diagnostic-invalid-utf8, clang-diagnostic-invalid-source-encoding, clang-diagnostic-pointer-arith, clang-diagnostic-strict-prototypes, hicpp-uppercase-literal-suffix, cppcoreguidelines-*, performance-*)

/* Addiert zwei Integer-Strings */
signed long BrbIntegerStringAdd(plcstring* pIntegerString1, plcstring* pIntegerString2, unsigned long nSize1)
{
	if(pIntegerString1 == 0 || pIntegerString2 == 0)
	{
		return eBRB_ERR_NULL_POINTER;
	}
	UDINT nLen1 = strlen(pIntegerString1);
	UDINT nLen2 = strlen(pIntegerString2);
	UDINT nLenMax = nLen1;
	if(nLen2 > nLen1)
	{
		nLenMax = nLen2;
	}
	// Temporärer Ergebnis-String
	STRING sResult[nSize1];
	memset((USINT*)&sResult, 0 ,sizeof(sResult));
	BrbStringPadRight(sResult, "0", nSize1-1);
	// Stellen des längsten Strings von hinten nach vorne durchgehen
	UDINT nDigit = 0; // Stelle von hinten
	BOOL bDigitOverflow = 0;
	for(nDigit=0; nDigit<nLenMax+1; nDigit++) // nLenMax+1, damit der Überlauf der letzten Stelle auch berücksichtigt wird
	{
		// Stellenwert von String1 ermitteln
		USINT nValue1 = 0;
		if(nDigit < nLen1)
		{
			USINT* pChar1 = (USINT*)pIntegerString1 + nLen1 - nDigit - 1;
			nValue1 = *pChar1 - '0';
		}
		// Stellenwert von String2 ermitteln
		USINT nValue2 = 0;
		if(nDigit < nLen2)
		{
			USINT* pChar2 = (USINT*)pIntegerString2 + nLen2 - nDigit - 1;
			nValue2 = *pChar2 - '0';
		}
		// Summe ermitteln
		USINT nSum = nValue1 + nValue2;
		if(bDigitOverflow == 1)
		{
			// Überlauf aus vorherigem Durchgang berücksichtigen
			nSum += 1;
			bDigitOverflow = 0;
		}
		// Überlauf ermitteln
		if(nSum >= 10)
		{
			nSum -= 10;
			bDigitOverflow = 1;
		}
		if(nDigit < nSize1)
		{
			// Summe in Ergebnis besetzen
			USINT* pCharResult = (USINT*)&sResult + nSize1 - nDigit - 2;
			*pCharResult = '0' + nSum;
		}
		else
		{
			// Ergebnis-String ist zu Ende -> Schleife verlassen
			break;
		}
	}
	// Ergebnis auf String1 übernehmen
	BrbStringTrimLeft(sResult, "0");
	if(strlen(sResult) == 0)
	{
		BrbStringCopy(sResult, "0", nSize1);
	}
	BrbStringCopy(pIntegerString1, sResult, nSize1);
	return eBRB_ERR_OK;
}

// NOLINTEND(readability-*, bugprone-easily-swappable-parameters, clang-diagnostic-invalid-utf8, clang-diagnostic-invalid-source-encoding, clang-diagnostic-pointer-arith, clang-diagnostic-strict-prototypes, hicpp-uppercase-literal-suffix, cppcoreguidelines-*, performance-*)
```

#### BrbByteArrayAdd.c
```c
#include <bur/plctypes.h>
#ifdef __cplusplus
	extern "C"
	{
#endif

#include "BrbLib.h"

#ifdef __cplusplus
	};
#endif

// NOLINTBEGIN(readability-*, bugprone-easily-swappable-parameters, clang-diagnostic-invalid-utf8, clang-diagnostic-invalid-source-encoding, clang-diagnostic-pointer-arith, clang-diagnostic-strict-prototypes, hicpp-uppercase-literal-suffix, cppcoreguidelines-*, performance-*)

/* Addiert zwei Zahlen, welche als Byte-Array abgelegt sind */
signed long BrbByteArrayAdd(unsigned char* pByteArray0, unsigned long nLength0, unsigned char* pByteArray1, unsigned long nLength1)
{
	if(pByteArray0 == 0 || pByteArray1 == 0)
	{
		return eBRB_ERR_NULL_POINTER;
	}
	UDINT nLength = nLength0;
	if(nLength1 > nLength0)
	{
		nLength = nLength1;
	}
	UDINT nBitNumberMax = nLength * nBRB_BITS_PER_BYTE;
	UDINT nBitNumber = 0;
	BOOL bBitOverflow = 0;
	for(nBitNumber=0; nBitNumber<nBitNumberMax; nBitNumber++)
	{
		BOOL bBitValue0 = BrbGetByteArrayBit((UDINT)pByteArray0, nBitNumberMax, nBitNumber);
		BOOL bBitValue1 = BrbGetByteArrayBit((UDINT)pByteArray1, nBitNumberMax, nBitNumber);
		BOOL bBitResult = bBitValue0 ^ bBitValue1; // XOR rechnet beide Operanden
		bBitResult = bBitResult ^ bBitOverflow; // XOR rechnet Overflow ein
		BrbSetByteArrayBit((UDINT)pByteArray0, nBitNumberMax, nBitNumber, bBitResult);
		USINT nOverflow = (USINT)bBitValue0 + (USINT)bBitValue1 + (USINT)bBitOverflow;
		// Overflow für die nächste Stelle ermitteln
		bBitOverflow = 0;
		if(nOverflow > 1)
		{
			// Mehr als 1 Bit gesetzt -> Overflow für die nächste Stelle
			bBitOverflow = 1;
		}
	}
	if(bBitOverflow == 1)
	{
		return eBRB_ERR_OVERFLOW;
	}
	return eBRB_ERR_OK;
}

// NOLINTEND(readability-*, bugprone-easily-swappable-parameters, clang-diagnostic-invalid-utf8, clang-diagnostic-invalid-source-encoding, clang-diagnostic-pointer-arith, clang-diagnostic-strict-prototypes, hicpp-uppercase-literal-suffix, cppcoreguidelines-*, performance-*)
```

#### BrbByteArraySubtract.c
```c
#include <bur/plctypes.h>
#ifdef __cplusplus
	extern "C"
	{
#endif

#include "BrbLib.h"

#ifdef __cplusplus
	};
#endif

// NOLINTBEGIN(readability-*, bugprone-easily-swappable-parameters, clang-diagnostic-invalid-utf8, clang-diagnostic-invalid-source-encoding, clang-diagnostic-pointer-arith, clang-diagnostic-strict-prototypes, hicpp-uppercase-literal-suffix, cppcoreguidelines-*, performance-*)

/* Subtrahiert zwei Zahlen, welche als Byte-Array abgelegt sind */
signed long BrbByteArraySubtract(unsigned char* pByteArray0, unsigned long nLength0, unsigned char* pByteArray1, unsigned long nLength1)
{
	if(pByteArray0 == 0 || pByteArray1 == 0)
	{
		return eBRB_ERR_NULL_POINTER;
	}
	UDINT nLength = nLength0;
	if(nLength1 > nLength0)
	{
		nLength = nLength1;
	}
	UDINT nBitNumberMax = nLength * nBRB_BITS_PER_BYTE;
	UDINT nBitNumber = 0;
	BOOL bBitOverflow = 0;
	for(nBitNumber=0; nBitNumber<nBitNumberMax; nBitNumber++)
	{
		BOOL bBitValue0 = BrbGetByteArrayBit((UDINT)pByteArray0, nBitNumberMax, nBitNumber);
		BOOL bBitValue1 = BrbGetByteArrayBit((UDINT)pByteArray1, nBitNumberMax, nBitNumber);
		SINT nResult = (SINT)bBitValue0 - (SINT)bBitValue1 - (SINT)bBitOverflow; // NOLINT(bugprone-narrowing-conversions, cppcoreguidelines-narrowing-conversions)
		BOOL bBitResult = 0;
		bBitOverflow = 0;
		if(nResult == 1)
		{
			bBitResult = 1;
		}
		else if(nResult == 0)
		{
			bBitResult = 0;
		}
		else if(nResult == -1)
		{
			bBitResult = 1;
			bBitOverflow = 1;
		}
		else
		{
			bBitResult = 0;
			bBitOverflow = 1;
		}
		BrbSetByteArrayBit((UDINT)pByteArray0, nBitNumberMax, nBitNumber, bBitResult);
	}
	if(bBitOverflow == 1)
	{
		return eBRB_ERR_OVERFLOW;
	}
	return eBRB_ERR_OK;
}

// NOLINTEND(readability-*, bugprone-easily-swappable-parameters, clang-diagnostic-invalid-utf8, clang-diagnostic-invalid-source-encoding, clang-diagnostic-pointer-arith, clang-diagnostic-strict-prototypes, hicpp-uppercase-literal-suffix, cppcoreguidelines-*, performance-*)
```

#### Package Logical/Libraries/BrbLib/Xml - Xml-Funktionen

#### BrbXmlGetNextTag.c
```c
/********************************************************************
 * COPYRIGHT -- Bernecker + Rainer
 ********************************************************************
 * Library: BrbLib
 * File: BrbXmlGetNextTag.c
 * Author: niedermeierr
 * Created: June 11, 2013
 ********************************************************************
 * Implementation of library BrbLib
 ********************************************************************/

#include <bur/plctypes.h>
#ifdef __cplusplus
	extern "C"
	{
#endif

#include "BrbLib.h"
#include <string.h>

#ifdef __cplusplus
	};
#endif

// NOLINTBEGIN(readability-*, bugprone-easily-swappable-parameters, clang-diagnostic-invalid-utf8, clang-diagnostic-invalid-source-encoding, clang-diagnostic-pointer-arith, clang-diagnostic-strict-prototypes, hicpp-uppercase-literal-suffix, cppcoreguidelines-*, performance-*)

/* Gibt die Adresse nach einem Xml-Tag zurück */
unsigned long BrbXmlGetNextTag(plcstring* pTag, unsigned long pStart, unsigned long pEnd)
{
	UDINT nResult = 0;
	// Start-Tag suchen
	STRING* pStartTagAdr = 0;
	if(pStart > 0 && pEnd > 0 && pEnd > pStart)
	{
		UDINT nSearchLen = pEnd - pStart;
		pStartTagAdr = BrbStringGetAdrOf((STRING*)pStart, pTag, nSearchLen);
		if(pStartTagAdr != 0)
		{
			// Start-Tag gefunden
			UDINT nStartTagLen = strlen(pTag);
			nResult = (UDINT)(pStartTagAdr + nStartTagLen);
		}
	}
	return nResult;
}

// NOLINTEND(readability-*, bugprone-easily-swappable-parameters, clang-diagnostic-invalid-utf8, clang-diagnostic-invalid-source-encoding, clang-diagnostic-pointer-arith, clang-diagnostic-strict-prototypes, hicpp-uppercase-literal-suffix, cppcoreguidelines-*, performance-*)
```

#### BrbXmlGetTagText.c
```c
/********************************************************************
 * COPYRIGHT -- Bernecker + Rainer
 ********************************************************************
 * Library: BrbLib
 * File: BrbXmlGetTagText.c
 * Author: niedermeierr
 * Created: June 11, 2013
 ********************************************************************
 * Implementation of library BrbLib
 ********************************************************************/

#include <bur/plctypes.h>
#ifdef __cplusplus
	extern "C"
	{
#endif

#include "BrbLib.h"
#include <string.h>

#ifdef __cplusplus
	};
#endif

// NOLINTBEGIN(readability-*, bugprone-easily-swappable-parameters, clang-diagnostic-invalid-utf8, clang-diagnostic-invalid-source-encoding, clang-diagnostic-pointer-arith, clang-diagnostic-strict-prototypes, hicpp-uppercase-literal-suffix, cppcoreguidelines-*, performance-*)

/* Gibt den Text zwischen zwei Xml-Tags zurück */
unsigned long BrbXmlGetTagText(plcstring* pStartTag, plcstring* pEndTag, unsigned long pStart, unsigned long pEnd, plcstring* pText, unsigned long nTextSize)
{
	UDINT nResult = 0;
	// Zu füllenden Text löschen
	memset(pText, 0, nTextSize);
	// Start-Tag suchen
	STRING* pStartTagAdr = 0;
	if(pStart > 0 && pEnd > 0 && pEnd > pStart)
	{
		UDINT nSearchLen = pEnd - pStart;
		pStartTagAdr = BrbStringGetAdrOf((STRING*)pStart, pStartTag, nSearchLen);
		if(pStartTagAdr != 0)
		{
			UDINT nStartTagLen = strlen(pStartTag);
			nResult = (UDINT)(pStartTagAdr + nStartTagLen);
			// Start-Tag gefunden -> End-Tag suchen
			STRING* pEndTagAdr = 0;
			pEndTagAdr = BrbStringGetAdrOf(pStartTagAdr, pEndTag, pEnd - (UDINT)pStartTagAdr);
			if(pEndTagAdr != 0)
			{
				// End-Tag gefunden -> Zeichen zwischen Start- und End-Tag durchtickern
				USINT* pCharSource = 0;
				UDINT nCharDestIndex = 0;
				for(pCharSource=(USINT*)pStartTagAdr + nStartTagLen; pCharSource<(USINT*)pEndTagAdr; pCharSource++)
				{
					// Nur Ascii-Zeichen übernehmen
					if((*pCharSource >= 32) && (*pCharSource <= 126))
					{
						USINT* pCharDest = (USINT*)pText + nCharDestIndex;
						*pCharDest = *pCharSource;
						nCharDestIndex += 1;
						if(nCharDestIndex >= nTextSize)
						{
							// Größe des zu füllenden Strings darf nicht überschritten werden
							break;
						}
					}
				}
				UDINT nEndTagLen = strlen(pEndTag);
				nResult = (UDINT)(pEndTagAdr + nEndTagLen);
			}
		}
	}
	return nResult;
}

// NOLINTEND(readability-*, bugprone-easily-swappable-parameters, clang-diagnostic-invalid-utf8, clang-diagnostic-invalid-source-encoding, clang-diagnostic-pointer-arith, clang-diagnostic-strict-prototypes, hicpp-uppercase-literal-suffix, cppcoreguidelines-*, performance-*)
```

#### Package Logical/Libraries/BrbLib/Memory - Speicherverwaltung

#### BrbMemListClear.c - Löscht die gesamte Liste
```c
/********************************************************************
 * COPYRIGHT -- Bernecker + Rainer
 ********************************************************************
 * Library: BrbLib
 * File: BrbMemListClear.c
 * Author: niedermeierr
 * Created: June 11, 2013
 ********************************************************************
 * Implementation of library BrbLib
 ********************************************************************/

#include <bur/plctypes.h>
#ifdef __cplusplus
	extern "C"
	{
#endif

#include "BrbLib.h"
#include <string.h>

#ifdef __cplusplus
	};
#endif

// NOLINTBEGIN(readability-*, bugprone-easily-swappable-parameters, clang-diagnostic-invalid-utf8, clang-diagnostic-invalid-source-encoding, clang-diagnostic-pointer-arith, clang-diagnostic-strict-prototypes, hicpp-uppercase-literal-suffix, cppcoreguidelines-*, performance-*)

/* Löscht die gesamte Liste */
signed long BrbMemListClear(struct BrbMemListManagement_Typ* pListManagement)
{
	DINT nResult = -1;
	if(pListManagement != 0)
	{
		if(pListManagement->pList > 0)
		{
			// Länge der Liste berechnen
			UDINT nLen = (pListManagement->nIndexMax+1) * pListManagement->nEntryLength;
			// Komplette Liste löschen
			memset((USINT*)pListManagement->pList, 0, nLen);
			// Anzahl auf 0 setzen
			pListManagement->nEntryCount = 0;
			nResult = 0;
		}
	}
	return nResult;
}

// NOLINTEND(readability-*, bugprone-easily-swappable-parameters, clang-diagnostic-invalid-utf8, clang-diagnostic-invalid-source-encoding, clang-diagnostic-pointer-arith, clang-diagnostic-strict-prototypes, hicpp-uppercase-literal-suffix, cppcoreguidelines-*, performance-*)
```

#### BrbMemListIn.c - Fügt einen Eintrag an bestimmter Stelle in der Liste ein
```c
/********************************************************************
 * COPYRIGHT -- Bernecker + Rainer
 ********************************************************************
 * Library: BrbLib
 * File: BrbMemListIn.c
 * Author: niedermeierr
 * Created: June 11, 2013
 ********************************************************************
 * Implementation of library BrbLib
 ********************************************************************/

#include <bur/plctypes.h>
#ifdef __cplusplus
	extern "C"
	{
#endif

#include "BrbLib.h"
#include <string.h>

#ifdef __cplusplus
	};
#endif

// NOLINTBEGIN(readability-*, bugprone-easily-swappable-parameters, clang-diagnostic-invalid-utf8, clang-diagnostic-invalid-source-encoding, clang-diagnostic-pointer-arith, clang-diagnostic-strict-prototypes, hicpp-uppercase-literal-suffix, cppcoreguidelines-*, performance-*)

/* Fügt einen Eintrag an bestimmter Stelle in der Liste ein */
signed long BrbMemListIn(struct BrbMemListManagement_Typ* pListManagement, unsigned long nIndex, unsigned long pNewEntry)
{
	DINT nResult = -1;
	if(pListManagement != 0)
	{
		if(pListManagement->pList > 0)
		{
			if(pNewEntry > 0)
			{
				// Prüfen, ob noch ein Platz frei ist
				if((pListManagement->nEntryCount == 0) || ((pListManagement->nEntryCount-1) < pListManagement->nIndexMax))
				{
					// Prüfen, ob Index gültig
					if(nIndex <= pListManagement->nEntryCount)
					{
						// Alle Einträge ab nIndex um 1 nach unten schieben
						UDINT pListSource = pListManagement->pList + (nIndex * pListManagement->nEntryLength);
						UDINT pListDestination = pListManagement->pList + ((nIndex+1) * pListManagement->nEntryLength);
						UDINT nLen = pListManagement->nEntryLength * (pListManagement->nIndexMax - nIndex);
						memmove((USINT*)pListDestination, (USINT*)pListSource, nLen);
						// Übergebenen Eintrag in die Liste kopieren
						pListDestination = pListManagement->pList + (nIndex * pListManagement->nEntryLength);
						memcpy((USINT*)pListDestination, (USINT*)pNewEntry, pListManagement->nEntryLength);
						// Anzahl inkrementieren
						pListManagement->nEntryCount += 1;
						nResult = (DINT)nIndex;
					}
				}
			}
		}
	}
	return nResult;
}

// NOLINTEND(readability-*, bugprone-easily-swappable-parameters, clang-diagnostic-invalid-utf8, clang-diagnostic-invalid-source-encoding, clang-diagnostic-pointer-arith, clang-diagnostic-strict-prototypes, hicpp-uppercase-literal-suffix, cppcoreguidelines-*, performance-*)
```

#### BrbMemListOut.c - Holt einen bestimmten Eintrag und löscht ihn aus der Liste
```c
/********************************************************************
 * COPYRIGHT -- Bernecker + Rainer
 ********************************************************************
 * Library: BrbLib
 * File: BrbMemListOut.c
 * Author: niedermeierr
 * Created: June 11, 2013
 ********************************************************************
 * Implementation of library BrbLib
 ********************************************************************/

#include <bur/plctypes.h>
#ifdef __cplusplus
	extern "C"
	{
#endif

#include "BrbLib.h"
#include <string.h>

#ifdef __cplusplus
	};
#endif

// NOLINTBEGIN(readability-*, bugprone-easily-swappable-parameters, clang-diagnostic-invalid-utf8, clang-diagnostic-invalid-source-encoding, clang-diagnostic-pointer-arith, clang-diagnostic-strict-prototypes, hicpp-uppercase-literal-suffix, cppcoreguidelines-*, performance-*)

/* Holt einen bestimmten Eintrag und löscht ihn aus der Liste */
signed long BrbMemListOut(struct BrbMemListManagement_Typ* pListManagement, unsigned long nIndex, unsigned long pListEntry)
{
	DINT nResult = -1;
	if(pListManagement != 0)
	{
		if(pListManagement->pList > 0)
		{
			// Prüfen, ob ein Eintrag vorhanden ist
			if(pListManagement->nEntryCount > nIndex)
			{
				UDINT pListSource = 0;
				UDINT pListDestination = 0;
				if(pListEntry > 0)
				{
					// Adresse des Eintrags berechnen
					pListSource = pListManagement->pList + (nIndex * pListManagement->nEntryLength);
					// Eintrag kopieren
					memcpy((USINT*)pListEntry, (USINT*)pListSource, pListManagement->nEntryLength);
				}
				// Anzahl dekrementieren
				pListManagement->nEntryCount -= 1;
				// Alle folgenden Einträge um 1 nach oben schieben
				pListDestination = pListManagement->pList + (nIndex * pListManagement->nEntryLength);
				pListSource = pListManagement->pList + ((nIndex+1) * pListManagement->nEntryLength);
				UDINT nLen = pListManagement->nEntryLength * (pListManagement->nIndexMax - nIndex);
				memmove((USINT*)pListDestination, (USINT*)pListSource, nLen);
				// Letzten Eintrag löschen
				pListDestination = pListManagement->pList + (pListManagement->nIndexMax * pListManagement->nEntryLength);
				memset((USINT*)pListDestination, 0, pListManagement->nEntryLength);
				nResult = (DINT)nIndex;
			}
		}
	}
	return nResult;
}

// NOLINTEND(readability-*, bugprone-easily-swappable-parameters, clang-diagnostic-invalid-utf8, clang-diagnostic-invalid-source-encoding, clang-diagnostic-pointer-arith, clang-diagnostic-strict-prototypes, hicpp-uppercase-literal-suffix, cppcoreguidelines-*, performance-*)
```

#### BrbMemListGetEntry.c - Holt einen bestimmten Eintrag aus der Liste
```c
/********************************************************************
 * COPYRIGHT -- Bernecker + Rainer
 ********************************************************************
 * Library: BrbLib
 * File: BrbMemListGetEntry.c
 * Author: niedermeierr
 * Created: June 11, 2013
 ********************************************************************
 * Implementation of library BrbLib
 ********************************************************************/

#include <bur/plctypes.h>
#ifdef __cplusplus
	extern "C"
	{
#endif

#include "BrbLib.h"
#include <string.h>

#ifdef __cplusplus
	};
#endif

// NOLINTBEGIN(readability-*, bugprone-easily-swappable-parameters, clang-diagnostic-invalid-utf8, clang-diagnostic-invalid-source-encoding, clang-diagnostic-pointer-arith, clang-diagnostic-strict-prototypes, hicpp-uppercase-literal-suffix, cppcoreguidelines-*, performance-*)

/* Holt einen bestimmten Eintrag aus der Liste */
signed long BrbMemListGetEntry(struct BrbMemListManagement_Typ* pListManagement, unsigned long nIndex, unsigned long pListEntry)
{
	DINT nResult = -1;
	if(pListManagement != 0)
	{
		if(pListManagement->pList > 0)
		{
			// Prüfen, ob ein Eintrag vorhanden ist
			if(pListManagement->nEntryCount > nIndex)
			{
				UDINT pListSource = 0;
				if(pListEntry > 0)
				{
					// Adresse des Eintrags berechnen
					pListSource = pListManagement->pList + (nIndex * pListManagement->nEntryLength);
					// Eintrag kopieren
					memcpy((USINT*)pListEntry, (USINT*)pListSource, pListManagement->nEntryLength);
				}
				nResult = (DINT)nIndex;
			}
		}
	}
	return nResult;
}

// NOLINTEND(readability-*, bugprone-easily-swappable-parameters, clang-diagnostic-invalid-utf8, clang-diagnostic-invalid-source-encoding, clang-diagnostic-pointer-arith, clang-diagnostic-strict-prototypes, hicpp-uppercase-literal-suffix, cppcoreguidelines-*, performance-*)
```

#### BrbFifoIn.c - Fügt einen neuen Eintrag an der letzten Stelle hinzu
```c
/********************************************************************
 * COPYRIGHT -- Bernecker + Rainer
 ********************************************************************
 * Library: BrbLib
 * File: BrbFifoIn.c
 * Author: niedermeierr
 * Created: June 11, 2013
 ********************************************************************
 * Implementation of library BrbLib
 ********************************************************************/

#include <bur/plctypes.h>
#ifdef __cplusplus
	extern "C"
	{
#endif

#include "BrbLib.h"

#ifdef __cplusplus
	};
#endif

// NOLINTBEGIN(readability-*, bugprone-easily-swappable-parameters, clang-diagnostic-invalid-utf8, clang-diagnostic-invalid-source-encoding, clang-diagnostic-pointer-arith, clang-diagnostic-strict-prototypes, hicpp-uppercase-literal-suffix, cppcoreguidelines-*, performance-*)

/* Fügt einen neuen Eintrag an der letzten Stelle hinzu */
signed long BrbFifoIn(struct BrbMemListManagement_Typ* pListManagement, unsigned long pNewEntry)
{
	if(pListManagement != 0)
	{
		return BrbMemListIn(pListManagement, pListManagement->nEntryCount, pNewEntry);
	}
	else
	{
		return -1;
	}
}

// NOLINTEND(readability-*, bugprone-easily-swappable-parameters, clang-diagnostic-invalid-utf8, clang-diagnostic-invalid-source-encoding, clang-diagnostic-pointer-arith, clang-diagnostic-strict-prototypes, hicpp-uppercase-literal-suffix, cppcoreguidelines-*, performance-*)
```

#### BrbFifoOut.c - Gibt den Eintrag an erster Stelle zurück und löscht ihn aus der Liste
```c
/********************************************************************
 * COPYRIGHT -- Bernecker + Rainer
 ********************************************************************
 * Library: BrbLib
 * File: BrbFifoOut.c
 * Author: niedermeierr
 * Created: June 11, 2013
 ********************************************************************
 * Implementation of library BrbLib
 ********************************************************************/

#include <bur/plctypes.h>
#ifdef __cplusplus
	extern "C"
	{
#endif

	#include "BrbLib.h"

#ifdef __cplusplus
	};
#endif

// NOLINTBEGIN(readability-*, bugprone-easily-swappable-parameters, clang-diagnostic-invalid-utf8, clang-diagnostic-invalid-source-encoding, clang-diagnostic-pointer-arith, clang-diagnostic-strict-prototypes, hicpp-uppercase-literal-suffix, cppcoreguidelines-*, performance-*)

/* Gibt den Eintrag an erster Stelle zurück und löscht ihn aus der Liste */
signed long BrbFifoOut(struct BrbMemListManagement_Typ* pListManagement, unsigned long pListEntry)
{
	DINT nResult = -1;
	if(pListManagement != 0)
	{
		if(pListManagement->nEntryCount > 0)
		{
			nResult = BrbMemListOut(pListManagement, 0, pListEntry);
		}
	}
	return nResult;
}

// NOLINTEND(readability-*, bugprone-easily-swappable-parameters, clang-diagnostic-invalid-utf8, clang-diagnostic-invalid-source-encoding, clang-diagnostic-pointer-arith, clang-diagnostic-strict-prototypes, hicpp-uppercase-literal-suffix, cppcoreguidelines-*, performance-*)
```

#### BrbLifoIn.c - Fügt einen neuen Eintrag an der letzten Stelle hinzu
```c
/********************************************************************
 * COPYRIGHT -- Bernecker + Rainer
 ********************************************************************
 * Library: BrbLib
 * File: BrbLifoIn.c
 * Author: niedermeierr
 * Created: June 11, 2013
 ********************************************************************
 * Implementation of library BrbLib
 ********************************************************************/

#include <bur/plctypes.h>
#ifdef __cplusplus
	extern "C"
	{
#endif

	#include "BrbLib.h"

#ifdef __cplusplus
	};
#endif

// NOLINTBEGIN(readability-*, bugprone-easily-swappable-parameters, clang-diagnostic-invalid-utf8, clang-diagnostic-invalid-source-encoding, clang-diagnostic-pointer-arith, clang-diagnostic-strict-prototypes, hicpp-uppercase-literal-suffix, cppcoreguidelines-*, performance-*)

/* Fügt einen neuen Eintrag an der letzten Stelle hinzu */
signed long BrbLifoIn(struct BrbMemListManagement_Typ* pListManagement, unsigned long pNewEntry)
{
	if(pListManagement != 0)
	{
		return BrbMemListIn(pListManagement, pListManagement->nEntryCount, pNewEntry);
	}
	else
	{
		return -1;
	}
}

// NOLINTEND(readability-*, bugprone-easily-swappable-parameters, clang-diagnostic-invalid-utf8, clang-diagnostic-invalid-source-encoding, clang-diagnostic-pointer-arith, clang-diagnostic-strict-prototypes, hicpp-uppercase-literal-suffix, cppcoreguidelines-*, performance-*)
```

#### BrbLifoOut.c - Gibt den Eintrag an letzter Stelle zurück und löscht ihn aus der Liste
```c
/********************************************************************
 * COPYRIGHT -- Bernecker + Rainer
 ********************************************************************
 * Library: BrbLib
 * File: BrbLifoOut.c
 * Author: niedermeierr
 * Created: June 11, 2013
 ********************************************************************
 * Implementation of library BrbLib
 ********************************************************************/

#include <bur/plctypes.h>
#ifdef __cplusplus
	extern "C"
	{
#endif

	#include "BrbLib.h"

#ifdef __cplusplus
	};
#endif

// NOLINTBEGIN(readability-*, bugprone-easily-swappable-parameters, clang-diagnostic-invalid-utf8, clang-diagnostic-invalid-source-encoding, clang-diagnostic-pointer-arith, clang-diagnostic-strict-prototypes, hicpp-uppercase-literal-suffix, cppcoreguidelines-*, performance-*)

/* Gibt den Eintrag an letzter Stelle zurück und löscht ihn aus der Liste */
signed long BrbLifoOut(struct BrbMemListManagement_Typ* pListManagement, unsigned long pListEntry)
{
	DINT nResult = -1;
	if(pListManagement != 0)
	{
		if(pListManagement->nEntryCount > 0)
		{
			nResult = BrbMemListOut(pListManagement, pListManagement->nEntryCount - 1, pListEntry);
		}
	}
	return nResult;
}

// NOLINTEND(readability-*, bugprone-easily-swappable-parameters, clang-diagnostic-invalid-utf8, clang-diagnostic-invalid-source-encoding, clang-diagnostic-pointer-arith, clang-diagnostic-strict-prototypes, hicpp-uppercase-literal-suffix, cppcoreguidelines-*, performance-*)
```

#### BrbGetBitUdint.c - Liest ein Bit aus einem Udint
```c
/********************************************************************
 * COPYRIGHT -- Bernecker + Rainer
 ********************************************************************
 * Library: BrbLib
 * File: BrbGetBitUdint.c
 * Author: niedermeierr
 * Created: June 25, 2013
 ********************************************************************
 * Implementation of library BrbLib
 ********************************************************************/

#include <bur/plctypes.h>
#ifdef __cplusplus
	extern "C"
	{
#endif

#include "BrbLib.h"

#ifdef __cplusplus
	};
#endif

// NOLINTBEGIN(readability-*, bugprone-easily-swappable-parameters, clang-diagnostic-invalid-utf8, clang-diagnostic-invalid-source-encoding, clang-diagnostic-pointer-arith, clang-diagnostic-strict-prototypes, hicpp-uppercase-literal-suffix, cppcoreguidelines-*, performance-*)

/* Liest ein Bit aus einem Udint */
plcbit BrbGetBitUdint(unsigned long nValue, unsigned short nBitNumber)
{
	BOOL bResult = 0;
	if(nBitNumber <= 31)
	{
		bResult = (nValue & ((UDINT)1 << nBitNumber)) > 0;
	}
	return bResult;
}

// NOLINTEND(readability-*, bugprone-easily-swappable-parameters, clang-diagnostic-invalid-utf8, clang-diagnostic-invalid-source-encoding, clang-diagnostic-pointer-arith, clang-diagnostic-strict-prototypes, hicpp-uppercase-literal-suffix, cppcoreguidelines-*, performance-*)
```

#### BrbSetBitUdint.c - Setzt ein Bit in einem Udint
```c
/********************************************************************
 * COPYRIGHT -- Bernecker + Rainer
 ********************************************************************
 * Library: BrbLib
 * File: BrbSetBitUdint.c
 * Author: niedermeierr
 * Created: June 25, 2013
 ********************************************************************
 * Implementation of library BrbLib
 ********************************************************************/

#include <bur/plctypes.h>
#ifdef __cplusplus
	extern "C"
	{
#endif

#include "BrbLib.h"

#ifdef __cplusplus
	};
#endif

// NOLINTBEGIN(readability-*, bugprone-easily-swappable-parameters, clang-diagnostic-invalid-utf8, clang-diagnostic-invalid-source-encoding, clang-diagnostic-pointer-arith, clang-diagnostic-strict-prototypes, hicpp-uppercase-literal-suffix, cppcoreguidelines-*, performance-*)

/* Setzt oder löscht ein Bit in einem Udint */
plcbit BrbSetBitUdint(unsigned long* pValue, unsigned short nBitNumber, plcbit bBit)
{
	BOOL bResult = 0;
	if(nBitNumber <= 31)
	{
		bResult = BrbGetBitUdint(*pValue, nBitNumber);
		if(bBit == 1)
		{
			*pValue = *pValue | ((UDINT)1 << nBitNumber);
		}
		else
		{
			*pValue = *pValue & ~((UDINT)1 << nBitNumber);
		}
	}
	return bResult;
}

// NOLINTEND(readability-*, bugprone-easily-swappable-parameters, clang-diagnostic-invalid-utf8, clang-diagnostic-invalid-source-encoding, clang-diagnostic-pointer-arith, clang-diagnostic-strict-prototypes, hicpp-uppercase-literal-suffix, cppcoreguidelines-*, performance-*)
```

#### BrbGetBitmaskUdint.c - Liest eine Bitmaske aus einem Udint
```c
/********************************************************************
 * COPYRIGHT -- Bernecker + Rainer
 ********************************************************************
 * Library: BrbLib
 * File: BrbGetBitMaskUdint.c
 * Author: niedermeierr
 * Created: May 16, 2014
 ********************************************************************
 * Implementation of library BrbLib
 ********************************************************************/

#include <bur/plctypes.h>
#ifdef __cplusplus
	extern "C"
	{
#endif

#include "BrbLib.h"

#ifdef __cplusplus
	};
#endif

// NOLINTBEGIN(readability-*, bugprone-easily-swappable-parameters, clang-diagnostic-invalid-utf8, clang-diagnostic-invalid-source-encoding, clang-diagnostic-pointer-arith, clang-diagnostic-strict-prototypes, hicpp-uppercase-literal-suffix, cppcoreguidelines-*, performance-*)

/* Liest eine Bitmaske aus einem Udint */
plcbit BrbGetBitMaskUdint(unsigned long nValue, unsigned long nBitMask)
{
	UDINT nTest = nValue & nBitMask;
	BOOL bResult = (nTest == nBitMask);
	return bResult;
}

// NOLINTEND(readability-*, bugprone-easily-swappable-parameters, clang-diagnostic-invalid-utf8, clang-diagnostic-invalid-source-encoding, clang-diagnostic-pointer-arith, clang-diagnostic-strict-prototypes, hicpp-uppercase-literal-suffix, cppcoreguidelines-*, performance-*)
```

#### BrbSetBitMaskUdint.c - Setzt oder löscht eine Bitmaske in einem Udint
```c
/********************************************************************
 * COPYRIGHT -- Bernecker + Rainer
 ********************************************************************
 * Library: BrbLib
 * File: BrbSetBitMaskUdint.c
 * Author: niedermeierr
 * Created: May 16, 2014
 ********************************************************************
 * Implementation of library BrbLib
 ********************************************************************/

#include <bur/plctypes.h>
#ifdef __cplusplus
	extern "C"
	{
#endif

#include "BrbLib.h"

#ifdef __cplusplus
	};
#endif

// NOLINTBEGIN(readability-*, bugprone-easily-swappable-parameters, clang-diagnostic-invalid-utf8, clang-diagnostic-invalid-source-encoding, clang-diagnostic-pointer-arith, clang-diagnostic-strict-prototypes, hicpp-uppercase-literal-suffix, cppcoreguidelines-*, performance-*)

/* Setzt oder löscht eine Bitmaske in einem Udint */
plcbit BrbSetBitMaskUdint(unsigned long* pValue, unsigned long nBitMask, plcbit bSet)
{
	BOOL bResult = 0;
	bResult = BrbGetBitMaskUdint(*pValue, nBitMask);
	if(bSet == 1)
	{
		*pValue = *pValue | nBitMask;
	}
	else
	{
		*pValue = *pValue & ~nBitMask;
	}
	return bResult;
}

// NOLINTEND(readability-*, bugprone-easily-swappable-parameters, clang-diagnostic-invalid-utf8, clang-diagnostic-invalid-source-encoding, clang-diagnostic-pointer-arith, clang-diagnostic-strict-prototypes, hicpp-uppercase-literal-suffix, cppcoreguidelines-*, performance-*)
```

#### BrbGetBitUint.c - Liest ein Bit aus einem Uint
```c
/********************************************************************
 * COPYRIGHT -- Bernecker + Rainer
 ********************************************************************
 * Library: BrbLib
 * File: BrbGetBitUint.c
 * Author: niedermeierr
 * Created: June 25, 2013
 ********************************************************************
 * Implementation of library BrbLib
 ********************************************************************/

#include <bur/plctypes.h>
#ifdef __cplusplus
	extern "C"
	{
#endif

#include "BrbLib.h"

#ifdef __cplusplus
	};
#endif

// NOLINTBEGIN(readability-*, bugprone-easily-swappable-parameters, clang-diagnostic-invalid-utf8, clang-diagnostic-invalid-source-encoding, clang-diagnostic-pointer-arith, clang-diagnostic-strict-prototypes, hicpp-uppercase-literal-suffix, cppcoreguidelines-*, performance-*)

/* Liest ein Bit aus einem Uint */
plcbit BrbGetBitUint(unsigned short nValue, unsigned short nBitNumber)
{
	BOOL bResult = 0;
	if(nBitNumber <= 15)
	{
		bResult = (nValue & ((UINT)1 << nBitNumber)) > 0; // NOLINT(hicpp-signed-bitwise)
	}
	return bResult;
}

// NOLINTEND(readability-*, bugprone-easily-swappable-parameters, clang-diagnostic-invalid-utf8, clang-diagnostic-invalid-source-encoding, clang-diagnostic-pointer-arith, clang-diagnostic-strict-prototypes, hicpp-uppercase-literal-suffix, cppcoreguidelines-*, performance-*)
```

#### BrbSetBitUint.c - Setzt ein Bit in einem Uint
```c
/********************************************************************
 * COPYRIGHT -- Bernecker + Rainer
 ********************************************************************
 * Library: BrbLib
 * File: BrbSetBitUint.c
 * Author: niedermeierr
 * Created: June 25, 2013
 ********************************************************************
 * Implementation of library BrbLib
 ********************************************************************/

#include <bur/plctypes.h>
#ifdef __cplusplus
	extern "C"
	{
#endif

#include "BrbLib.h"

#ifdef __cplusplus
	};
#endif

// NOLINTBEGIN(readability-*, bugprone-easily-swappable-parameters, clang-diagnostic-invalid-utf8, clang-diagnostic-invalid-source-encoding, clang-diagnostic-pointer-arith, clang-diagnostic-strict-prototypes, hicpp-uppercase-literal-suffix, cppcoreguidelines-*, performance-*)

/* Setzt oder löscht ein Bit in einem Uint */
plcbit BrbSetBitUint(unsigned short* pValue, unsigned short nBitNumber, plcbit bBit)
{
	BOOL bResult = 0;
	if(nBitNumber <= 15)
	{
		bResult = BrbGetBitUint(*pValue, nBitNumber);
		if(bBit == 1)
		{
			*pValue = (UINT)(*pValue | ((UINT)1 << nBitNumber)); // NOLINT(hicpp-signed-bitwise)
		}
		else
		{
			*pValue = (UINT)(*pValue & ~((UINT)1 << nBitNumber)); // NOLINT(hicpp-signed-bitwise)
		}
	}
	return bResult;
}

// NOLINTEND(readability-*, bugprone-easily-swappable-parameters, clang-diagnostic-invalid-utf8, clang-diagnostic-invalid-source-encoding, clang-diagnostic-pointer-arith, clang-diagnostic-strict-prototypes, hicpp-uppercase-literal-suffix, cppcoreguidelines-*, performance-*)
```

#### BrbGetBitmaskUint.c - Liest eine Bitmaske aus einem Uint
```c
/********************************************************************
 * COPYRIGHT -- Bernecker + Rainer
 ********************************************************************
 * Library: BrbLib
 * File: BrbGetBitMaskUint.c
 * Author: niedermeierr
 * Created: May 16, 2014
 ********************************************************************
 * Implementation of library BrbLib
 ********************************************************************/

#include <bur/plctypes.h>
#ifdef __cplusplus
	extern "C"
	{
#endif

#include "BrbLib.h"

#ifdef __cplusplus
	};
#endif

// NOLINTBEGIN(readability-*, bugprone-easily-swappable-parameters, clang-diagnostic-invalid-utf8, clang-diagnostic-invalid-source-encoding, clang-diagnostic-pointer-arith, clang-diagnostic-strict-prototypes, hicpp-uppercase-literal-suffix, cppcoreguidelines-*, performance-*)

/* Liest eine Bitmaske aus einem Uint */
plcbit BrbGetBitMaskUint(unsigned short nValue, unsigned short nBitMask)
{
	UINT nTest = nValue & nBitMask;
	BOOL bResult = (nTest == nBitMask);
	return bResult;
}

// NOLINTEND(readability-*, bugprone-easily-swappable-parameters, clang-diagnostic-invalid-utf8, clang-diagnostic-invalid-source-encoding, clang-diagnostic-pointer-arith, clang-diagnostic-strict-prototypes, hicpp-uppercase-literal-suffix, cppcoreguidelines-*, performance-*)
```

#### BrbSetBitmaskUint.c - Setzt oder löscht eine Bitmaske in einem Uint
```c
/********************************************************************
 * COPYRIGHT -- Bernecker + Rainer
 ********************************************************************
 * Library: BrbLib
 * File: BrbSetBitMaskUint.c
 * Author: niedermeierr
 * Created: May 16, 2014
 ********************************************************************
 * Implementation of library BrbLib
 ********************************************************************/

#include <bur/plctypes.h>
#ifdef __cplusplus
	extern "C"
	{
#endif

#include "BrbLib.h"

#ifdef __cplusplus
	};
#endif

// NOLINTBEGIN(readability-*, bugprone-easily-swappable-parameters, clang-diagnostic-invalid-utf8, clang-diagnostic-invalid-source-encoding, clang-diagnostic-pointer-arith, clang-diagnostic-strict-prototypes, hicpp-uppercase-literal-suffix, cppcoreguidelines-*, performance-*)

/* Setzt oder löscht eine Bitmaske in einem Uint */
plcbit BrbSetBitMaskUint(unsigned short* pValue, unsigned short nBitMask, plcbit bSet)
{
	BOOL bResult = 0;
	bResult = BrbGetBitMaskUint(*pValue, nBitMask);
	if(bSet == 1)
	{
		*pValue = *pValue | nBitMask;
	}
	else
	{
		*pValue = *pValue & ~nBitMask; // NOLINT(hicpp-signed-bitwise)
	}
	return bResult;
}

// NOLINTEND(readability-*, bugprone-easily-swappable-parameters, clang-diagnostic-invalid-utf8, clang-diagnostic-invalid-source-encoding, clang-diagnostic-pointer-arith, clang-diagnostic-strict-prototypes, hicpp-uppercase-literal-suffix, cppcoreguidelines-*, performance-*)
```

#### BrbGetBitUsint.c - Liest ein Bit aus einem Usint
```c
/********************************************************************
 * COPYRIGHT -- Bernecker + Rainer
 ********************************************************************
 * Library: BrbLib
 * File: BrbGetBitUsint.c
 * Author: niedermeierr
 * Created: June 25, 2013
 ********************************************************************
 * Implementation of library BrbLib
 ********************************************************************/

#include <bur/plctypes.h>
#ifdef __cplusplus
	extern "C"
	{
#endif

#include "BrbLib.h"

#ifdef __cplusplus
	};
#endif

// NOLINTBEGIN(readability-*, bugprone-easily-swappable-parameters, clang-diagnostic-invalid-utf8, clang-diagnostic-invalid-source-encoding, clang-diagnostic-pointer-arith, clang-diagnostic-strict-prototypes, hicpp-uppercase-literal-suffix, cppcoreguidelines-*, performance-*)

/* Liest ein Bit aus einem Usint */
plcbit BrbGetBitUsint(unsigned char nValue, unsigned short nBitNumber)
{
	BOOL bResult = 0;
	if(nBitNumber <= 7)
	{
		bResult = (nValue & ((USINT)1 << nBitNumber)) > 0; // NOLINT(hicpp-signed-bitwise)
	}
	return bResult;
}

// NOLINTEND(readability-*, bugprone-easily-swappable-parameters, clang-diagnostic-invalid-utf8, clang-diagnostic-invalid-source-encoding, clang-diagnostic-pointer-arith, clang-diagnostic-strict-prototypes, hicpp-uppercase-literal-suffix, cppcoreguidelines-*, performance-*)
```

#### BrbSetBitUsint.c - Setzt ein Bit in einem Usint
```c
/********************************************************************
 * COPYRIGHT -- Bernecker + Rainer
 ********************************************************************
 * Library: BrbLib
 * File: BrbSetBitUsint.c
 * Author: niedermeierr
 * Created: June 25, 2013
 ********************************************************************
 * Implementation of library BrbLib
 ********************************************************************/

#include <bur/plctypes.h>
#ifdef __cplusplus
	extern "C"
	{
#endif

#include "BrbLib.h"

#ifdef __cplusplus
	};
#endif

// NOLINTBEGIN(readability-*, bugprone-easily-swappable-parameters, clang-diagnostic-invalid-utf8, clang-diagnostic-invalid-source-encoding, clang-diagnostic-pointer-arith, clang-diagnostic-strict-prototypes, hicpp-uppercase-literal-suffix, cppcoreguidelines-*, performance-*)

/* Setzt ein Bit in einem Usint */
plcbit BrbSetBitUsint(unsigned char* pValue, unsigned short nBitNumber, plcbit bBit)
{
	BOOL bResult = 0;
	if(nBitNumber <= 7)
	{
		bResult = BrbGetBitUsint(*pValue, nBitNumber);
		if(bBit == 1)
		{
			*pValue = *pValue | (USINT)((USINT)1 << nBitNumber); // NOLINT(hicpp-signed-bitwise)
		}
		else
		{
			*pValue = *pValue & ~(USINT)((USINT)1 << nBitNumber); // NOLINT(hicpp-signed-bitwise)
		}
	}
	return bResult;
}

// NOLINTEND(readability-*, bugprone-easily-swappable-parameters, clang-diagnostic-invalid-utf8, clang-diagnostic-invalid-source-encoding, clang-diagnostic-pointer-arith, clang-diagnostic-strict-prototypes, hicpp-uppercase-literal-suffix, cppcoreguidelines-*, performance-*)
```

#### BrbGetBitmaskUsint.c - Liest eine Bitmaske aus einem Usint
```c
/********************************************************************
 * COPYRIGHT -- Bernecker + Rainer
 ********************************************************************
 * Library: BrbLib
 * File: BrbGetBitMaskUsint.c
 * Author: niedermeierr
 * Created: May 16, 2014
 ********************************************************************
 * Implementation of library BrbLib
 ********************************************************************/

#include <bur/plctypes.h>
#ifdef __cplusplus
	extern "C"
	{
#endif

#include "BrbLib.h"

#ifdef __cplusplus
	};
#endif

// NOLINTBEGIN(readability-*, bugprone-easily-swappable-parameters, clang-diagnostic-invalid-utf8, clang-diagnostic-invalid-source-encoding, clang-diagnostic-pointer-arith, clang-diagnostic-strict-prototypes, hicpp-uppercase-literal-suffix, cppcoreguidelines-*, performance-*)

/* Liest eine Bitmaske aus einem Usint */
plcbit BrbGetBitMaskUsint(unsigned char nValue, unsigned char nBitMask)
{
	USINT nTest = nValue & nBitMask;
	BOOL bResult = (nTest == nBitMask);
	return bResult;
}

// NOLINTEND(readability-*, bugprone-easily-swappable-parameters, clang-diagnostic-invalid-utf8, clang-diagnostic-invalid-source-encoding, clang-diagnostic-pointer-arith, clang-diagnostic-strict-prototypes, hicpp-uppercase-literal-suffix, cppcoreguidelines-*, performance-*)
```

#### BrbSetBitMaskUsint.c - Setzt oder löscht eine Bitmaske in einem Usint
```c
/********************************************************************
 * COPYRIGHT -- Bernecker + Rainer
 ********************************************************************
 * Library: BrbLib
 * File: BrbSetBitMaskUsint.c
 * Author: niedermeierr
 * Created: May 16, 2014
 ********************************************************************
 * Implementation of library BrbLib
 ********************************************************************/

#include <bur/plctypes.h>
#ifdef __cplusplus
	extern "C"
	{
#endif

#include "BrbLib.h"

#ifdef __cplusplus
	};
#endif

// NOLINTBEGIN(readability-*, bugprone-easily-swappable-parameters, clang-diagnostic-invalid-utf8, clang-diagnostic-invalid-source-encoding, clang-diagnostic-pointer-arith, clang-diagnostic-strict-prototypes, hicpp-uppercase-literal-suffix, cppcoreguidelines-*, performance-*)

/* Setzt oder löscht eine Bitmaske in einem Usint */
plcbit BrbSetBitMaskUsint(unsigned char* pValue, unsigned char nBitMask, plcbit bSet)
{
	BOOL bResult = 0;
	bResult = BrbGetBitMaskUsint(*pValue, nBitMask);
	if(bSet == 1)
	{
		*pValue = *pValue | nBitMask;
	}
	else
	{
		*pValue = *pValue & ~nBitMask; // NOLINT(hicpp-signed-bitwise)
	}
	return bResult;
}

// NOLINTEND(readability-*, bugprone-easily-swappable-parameters, clang-diagnostic-invalid-utf8, clang-diagnostic-invalid-source-encoding, clang-diagnostic-pointer-arith, clang-diagnostic-strict-prototypes, hicpp-uppercase-literal-suffix, cppcoreguidelines-*, performance-*)
```

#### BrbGetByteArrayBit.c - Gibt ein Bit eines Byte-Arrays zurück
```c
#include <bur/plctypes.h>
#ifdef __cplusplus
	extern "C"
	{
#endif

#include "BrbLib.h"

#ifdef __cplusplus
	};
#endif

// NOLINTBEGIN(readability-*, bugprone-easily-swappable-parameters, clang-diagnostic-invalid-utf8, clang-diagnostic-invalid-source-encoding, clang-diagnostic-pointer-arith, clang-diagnostic-strict-prototypes, hicpp-uppercase-literal-suffix, cppcoreguidelines-*, performance-*)

/* Gibt ein Bit eines bitcodierten Byte-Arrays zurück */
plcbit BrbGetByteArrayBit(unsigned long pByteArray, unsigned long nIndexMax, unsigned long nBitNumber)
{
	BOOL bResult = 0;
	if(pByteArray != 0)
	{
		UINT nByteIndex = (UINT)(nBitNumber / nBRB_BITS_PER_BYTE);
		if(nByteIndex <= nIndexMax)
		{
			UINT nByteBitNumber = (UINT)(nBitNumber - (nByteIndex * nBRB_BITS_PER_BYTE));
			USINT* pByte = ((USINT*)pByteArray) + nByteIndex;
			bResult = (*pByte & ((USINT)1 << nByteBitNumber)) > 0; // NOLINT(hicpp-signed-bitwise)
		}
	}
	return bResult;
}

// NOLINTEND(readability-*, bugprone-easily-swappable-parameters, clang-diagnostic-invalid-utf8, clang-diagnostic-invalid-source-encoding, clang-diagnostic-pointer-arith, clang-diagnostic-strict-prototypes, hicpp-uppercase-literal-suffix, cppcoreguidelines-*, performance-*)
```

#### BrbSetByteArrayBit.c - Setzt ein Bit eines Byte-Arrays
```c
#include <bur/plctypes.h>
#ifdef __cplusplus
	extern "C"
	{
#endif

	#include "BrbLib.h"

#ifdef __cplusplus
	};
#endif

// NOLINTBEGIN(readability-*, bugprone-easily-swappable-parameters, clang-diagnostic-invalid-utf8, clang-diagnostic-invalid-source-encoding, clang-diagnostic-pointer-arith, clang-diagnostic-strict-prototypes, hicpp-uppercase-literal-suffix, cppcoreguidelines-*, performance-*)

/* Setzt ein Bit in einem bitcodierten Byte-Array */
plcbit BrbSetByteArrayBit(unsigned long pByteArray, unsigned long nIndexMax, unsigned long nBitNumber, plcbit bBit)
{
	BOOL bResult = 0;
	if(pByteArray != 0)
	{
		UINT nByteIndex = (UINT)(nBitNumber / nBRB_BITS_PER_BYTE);
		if(nByteIndex <= nIndexMax)
		{
			UINT nByteBitNumber = (UINT)(nBitNumber - ((UDINT)nByteIndex * (UDINT)nBRB_BITS_PER_BYTE));
			USINT* pByte = ((USINT*)pByteArray) + nByteIndex;
			bResult = (*pByte & ((USINT)1 << nByteBitNumber)) > 0; // NOLINT(hicpp-signed-bitwise)
			if(bBit == 1)
			{
				*pByte = *pByte | (USINT)((USINT)1 << nByteBitNumber); // NOLINT(hicpp-signed-bitwise)
			}
			else
			{
				*pByte = *pByte & ~(USINT)((USINT)1 << nByteBitNumber); // NOLINT(hicpp-signed-bitwise)
			}
		}
	}
	return bResult;
}

// NOLINTEND(readability-*, bugprone-easily-swappable-parameters, clang-diagnostic-invalid-utf8, clang-diagnostic-invalid-source-encoding, clang-diagnostic-pointer-arith, clang-diagnostic-strict-prototypes, hicpp-uppercase-literal-suffix, cppcoreguidelines-*, performance-*)
```

#### BrbSetByteArrayBits.c - Setzt mehrere Bits eines Byte-Arrays
```c
#include <bur/plctypes.h>
#ifdef __cplusplus
	extern "C"
	{
#endif

#include "BrbLib.h"

#ifdef __cplusplus
	};
#endif

// NOLINTBEGIN(readability-*, bugprone-easily-swappable-parameters, clang-diagnostic-invalid-utf8, clang-diagnostic-invalid-source-encoding, clang-diagnostic-pointer-arith, clang-diagnostic-strict-prototypes, hicpp-uppercase-literal-suffix, cppcoreguidelines-*, performance-*)

/* Setzte Bits in einem bitcodierten Byte-Array */
plcbit BrbSetByteArrayBits(unsigned long pByteArray, unsigned long nIndexMax, unsigned long nBitNumberFrom, unsigned long nBitNumberTo, plcbit bBit)
{
	if(pByteArray != 0)
	{
		if(nBitNumberTo < nBitNumberFrom)
		{
			UDINT nHelp = nBitNumberTo;
			nBitNumberTo = nBitNumberFrom;
			nBitNumberFrom = nHelp;
		}
		UDINT nBitNumber = 0;
		for(nBitNumber=nBitNumberFrom; nBitNumber<=nBitNumberTo; nBitNumber++)
		{
			UINT nByteIndex = (UINT)(nBitNumber / nBRB_BITS_PER_BYTE);
			if(nByteIndex <= nIndexMax)
			{
				UINT nByteBitNumber = (UINT)(nBitNumber - ((UDINT)nByteIndex * (UDINT)nBRB_BITS_PER_BYTE));
				USINT* pByte = ((USINT*)pByteArray) + nByteIndex;
				if(bBit == 1)
				{
					*pByte = *pByte | (USINT)((USINT)1 << nByteBitNumber); // NOLINT(hicpp-signed-bitwise)
				}
				else
				{
					*pByte = *pByte & ~(USINT)((USINT)1 << nByteBitNumber); // NOLINT(hicpp-signed-bitwise)
				}
			}
			else
			{
				break;
			}
		}
	}
	return bBit;
}

// NOLINTEND(readability-*, bugprone-easily-swappable-parameters, clang-diagnostic-invalid-utf8, clang-diagnostic-invalid-source-encoding, clang-diagnostic-pointer-arith, clang-diagnostic-strict-prototypes, hicpp-uppercase-literal-suffix, cppcoreguidelines-*, performance-*)
```

#### Package Logical/Libraries/BrbLib/Math - Mathematische Funktionen

#### BrbAbsReal.c - Gibt den Absolut-Wert zurück
```c
#include <bur/plctypes.h>
#ifdef __cplusplus
	extern "C"
	{
#endif

#include "BrbLib.h"

#ifdef __cplusplus
	};
#endif

// NOLINTBEGIN(readability-*, bugprone-easily-swappable-parameters, clang-diagnostic-invalid-utf8, clang-diagnostic-invalid-source-encoding, clang-diagnostic-pointer-arith, clang-diagnostic-strict-prototypes, hicpp-uppercase-literal-suffix, cppcoreguidelines-*, performance-*)

/* Gibt den absoluten Wert zurück */
float BrbAbsReal(float rValue)
{
	REAL rResult = rValue;
	if(rValue < 0.0f)
	{
		rResult = rValue * -1.0f;
	}
	return rResult;
}

// NOLINTEND(readability-*, bugprone-easily-swappable-parameters, clang-diagnostic-invalid-utf8, clang-diagnostic-invalid-source-encoding, clang-diagnostic-pointer-arith, clang-diagnostic-strict-prototypes, hicpp-uppercase-literal-suffix, cppcoreguidelines-*, performance-*)
```

#### BrbAbsLReal.c - Gibt den Absolut-Wert zurück
```c
#include <bur/plctypes.h>
#ifdef __cplusplus
	extern "C"
	{
#endif

#include "BrbLib.h"

#ifdef __cplusplus
	};
#endif

// NOLINTBEGIN(readability-*, bugprone-easily-swappable-parameters, clang-diagnostic-invalid-utf8, clang-diagnostic-invalid-source-encoding, clang-diagnostic-pointer-arith, clang-diagnostic-strict-prototypes, hicpp-uppercase-literal-suffix, cppcoreguidelines-*, performance-*)

/* Gibt den absoluten Wert zurück */
double BrbAbsLReal(double rValue)
{
	LREAL rResult = rValue;
	if(rValue < 0.0)
	{
		rResult = rValue * -1.0;
	}
	return rResult;
}

// NOLINTEND(readability-*, bugprone-easily-swappable-parameters, clang-diagnostic-invalid-utf8, clang-diagnostic-invalid-source-encoding, clang-diagnostic-pointer-arith, clang-diagnostic-strict-prototypes, hicpp-uppercase-literal-suffix, cppcoreguidelines-*, performance-*)
```

#### BrbIsNearlyZeroReal.c - Gibt zurück, ob sich der Wert als 0 interpretieren lässt
```c
#include <bur/plctypes.h>
#ifdef __cplusplus
	extern "C"
	{
#endif

	#include "BrbLib.h"
	#include <AnsiCFunc.h>

#ifdef __cplusplus
	};
#endif

// NOLINTBEGIN(readability-*, bugprone-easily-swappable-parameters, clang-diagnostic-invalid-utf8, clang-diagnostic-invalid-source-encoding, clang-diagnostic-pointer-arith, clang-diagnostic-strict-prototypes, hicpp-uppercase-literal-suffix, cppcoreguidelines-*, performance-*)

/* Gibt zurück, ob ein REAL-Wert annähernd 0 ist */
plcbit BrbIsNearlyZeroReal(float rValue, float rTolerance)
{
	BOOL bResult = 0;
	if(rTolerance < 0.0f)
	{
		rTolerance = rTolerance * -1.00000000000f;
	}
	REAL rMin = -rTolerance;
	REAL rMax = rTolerance;
	if(rValue >= rMin && rValue <= rMax)
	{
		bResult = 1;
	}
	return bResult;
}

// NOLINTEND(readability-*, bugprone-easily-swappable-parameters, clang-diagnostic-invalid-utf8, clang-diagnostic-invalid-source-encoding, clang-diagnostic-pointer-arith, clang-diagnostic-strict-prototypes, hicpp-uppercase-literal-suffix, cppcoreguidelines-*, performance-*)
```

#### BrbIsNearlyZeroLReal.c - Gibt zurück, ob sich der Wert als 0 interpretieren lässt
```c
#include <bur/plctypes.h>
#ifdef __cplusplus
	extern "C"
	{
#endif

	#include "BrbLib.h"
	#include <AnsiCFunc.h>

#ifdef __cplusplus
	};
#endif

// NOLINTBEGIN(readability-*, bugprone-easily-swappable-parameters, clang-diagnostic-invalid-utf8, clang-diagnostic-invalid-source-encoding, clang-diagnostic-pointer-arith, clang-diagnostic-strict-prototypes, hicpp-uppercase-literal-suffix, cppcoreguidelines-*, performance-*)

/* Gibt zurück, ob ein LREAL-Wert annähernd 0 ist */
plcbit BrbIsNearlyZeroLReal(double rValue, double rTolerance)
{
	BOOL bResult = 0;
	if(rTolerance < 0.0)
	{
		rTolerance = rTolerance*(LREAL)-1.00000000000000000000;
	}
	LREAL rMin = -rTolerance;
	LREAL rMax = rTolerance;
	if(rValue >= rMin && rValue <= rMax)
	{
		bResult = 1;
	}
	return bResult;
}

// NOLINTEND(readability-*, bugprone-easily-swappable-parameters, clang-diagnostic-invalid-utf8, clang-diagnostic-invalid-source-encoding, clang-diagnostic-pointer-arith, clang-diagnostic-strict-prototypes, hicpp-uppercase-literal-suffix, cppcoreguidelines-*, performance-*)
```

#### BrbCompareReal.c
```c
#include <bur/plctypes.h>
#ifdef __cplusplus
	extern "C"
	{
#endif

#include "BrbLib.h"
#include "limits.h"
#include <math.h>

#ifdef __cplusplus
	};
#endif

// NOLINTBEGIN(readability-*, bugprone-easily-swappable-parameters, clang-diagnostic-invalid-utf8, clang-diagnostic-invalid-source-encoding, clang-diagnostic-pointer-arith, clang-diagnostic-strict-prototypes, hicpp-uppercase-literal-suffix, cppcoreguidelines-*, performance-*)

/* Vergleicht zwei REAL-Werte */
signed short BrbCompareReal(float rValue1, float rValue2)
{
	// Union zur Interpretation der verschiedenen Datentypen
	typedef union
	{
		REAL rReal;
		DINT nDint;
		UDINT nUdint;

	} BrbValueUnion_TYP;
	BrbValueUnion_TYP	Value1 = {}; // NOLINT(clang-diagnostic-gnu-empty-initializer)
	BrbValueUnion_TYP	Value2 = {}; // NOLINT(clang-diagnostic-gnu-empty-initializer)

	// Werte wandeln in Union
	Value1.rReal = rValue1;
	Value2.rReal = rValue2;

	// NAN (Not A Number = Keine Zahl) oder INF (Infinity = Unendlich)
	if((isnan(Value1.rReal) != 0) ||
		(isinf(Value1.rReal) != 0))
	{
		return(nBRB_INT_MIN);
	}
	if((isnan(Value2.rReal) != 0) ||
		(isinf(Value2.rReal) != 0))
	{
		return(nBRB_INT_MAX);
	}

	// Behandlung Werte = -0.0
	if(Value1.nUdint == 0x80000000)
	{
		Value1.nUdint = 0;
	}
	if(Value2.nUdint == 0x80000000)
	{
		Value2.nUdint = 0;
	}

	// Vorzeichen unterschiedlich?
	if((Value1.nDint < 0) != (Value2.nDint < 0))
	{
		return (INT)(((Value1.nDint >= 0) ? 1 : -1));
	}

	// Werte haben das gleiche Vorzeichen
	// Werte negativ?
	if(Value1.nDint < 0)
	{
		// Werte positiv wandeln
		Value1.nUdint = -Value1.nUdint;
		Value2.nUdint = -Value2.nUdint;
	}

	// Werte vergleichen
	return (INT)((Value1.nUdint > Value2.nUdint) - (Value1.nUdint < Value2.nUdint));
}

// NOLINTEND(readability-*, bugprone-easily-swappable-parameters, clang-diagnostic-invalid-utf8, clang-diagnostic-invalid-source-encoding, clang-diagnostic-pointer-arith, clang-diagnostic-strict-prototypes, hicpp-uppercase-literal-suffix, cppcoreguidelines-*, performance-*)
```

#### BrbCompareLReal.c
```c
#include <bur/plctypes.h>
#ifdef __cplusplus
	extern "C"
	{
#endif

#include "BrbLib.h"
#include "limits.h"
#include <math.h>

#ifdef __cplusplus
	};
#endif

#define LINT          signed long long
#define ULINT         unsigned long long

// NOLINTBEGIN(readability-*, bugprone-easily-swappable-parameters, clang-diagnostic-invalid-utf8, clang-diagnostic-invalid-source-encoding, clang-diagnostic-pointer-arith, clang-diagnostic-strict-prototypes, hicpp-uppercase-literal-suffix, cppcoreguidelines-*, performance-*)

/* Vergleicht zwei LREAL-Werte */
signed short BrbCompareLReal(double rValue1, double rValue2)
{
	// Union zur Interpretation der verschiedenen Datentypen
	typedef union
	{
		LREAL rLreal;
		LINT nLint;
		ULINT nUlint;

	} BrbValueUnion_TYP;
	BrbValueUnion_TYP	Value1 = {}; // NOLINT(clang-diagnostic-gnu-empty-initializer)
	BrbValueUnion_TYP	Value2 = {}; // NOLINT(clang-diagnostic-gnu-empty-initializer)

	// Werte wandeln in Union
	Value1.rLreal = rValue1;
	Value2.rLreal = rValue2;

	// NAN (Not A Number = Keine Zahl) oder INF (Infinity = Unendlich)
	if((isnan(Value1.rLreal) != 0) ||
		(isinf(Value1.rLreal) != 0))
	{
		return(nBRB_INT_MIN);
	}
	if((isnan(Value2.rLreal) != 0) ||
		(isinf(Value2.rLreal) != 0))
	{
		return(nBRB_INT_MAX);
	}

	// Behandlung Werte = -0.0
	if(Value1.nUlint == 0x8000000000000000LL)
	{
		Value1.nUlint = 0;
	}
	if(Value2.nUlint == 0x8000000000000000LL)
	{
		Value2.nUlint = 0;
	}

	// Vorzeichen unterschiedlich?
	if((Value1.nLint < 0) != (Value2.nLint < 0))
	{
		return (INT)(((Value1.nLint >= 0) ? 1 : -1));
	}

	// Werte haben das gleiche Vorzeichen
	// Werte negativ?
	if(Value1.nLint < 0)
	{
		// Werte positiv wandeln
		Value1.nUlint = -Value1.nUlint;
		Value2.nUlint = -Value2.nUlint;
	}

	// Werte vergleichen
	return (INT)((Value1.nUlint > Value2.nUlint) - (Value1.nUlint < Value2.nUlint));
}

// NOLINTEND(readability-*, bugprone-easily-swappable-parameters, clang-diagnostic-invalid-utf8, clang-diagnostic-invalid-source-encoding, clang-diagnostic-pointer-arith, clang-diagnostic-strict-prototypes, hicpp-uppercase-literal-suffix, cppcoreguidelines-*, performance-*)
```

#### BrbIsWithinRangeDint.c - Gibt zurück, ob sich ein Wert innerhalb eines Bereichs befindet
```c
#include <bur/plctypes.h>
#ifdef __cplusplus
	extern "C"
	{
#endif

	#include "BrbLib.h"
	#include <AnsiCFunc.h>

#ifdef __cplusplus
	};
#endif

// NOLINTBEGIN(readability-*, bugprone-easily-swappable-parameters, clang-diagnostic-invalid-utf8, clang-diagnostic-invalid-source-encoding, clang-diagnostic-pointer-arith, clang-diagnostic-strict-prototypes, hicpp-uppercase-literal-suffix, cppcoreguidelines-*, performance-*)

/* Gibt zurück, ob sich ein Wert innerhalb eines Bereichs befindet */
plcbit BrbIsWithinRangeDint(signed long nValue, signed long nRangeMin, signed long nRangeMax, signed long nTolerance)
{
	BOOL bResult = 0;
	if(nRangeMin > nRangeMax)
	{
		DINT nTemp = nRangeMin;
		nRangeMin = nRangeMax;
		nRangeMax = nTemp;
	}
	if(nTolerance < 0)
	{
		nTolerance = abs(nTolerance);
	}
	DINT nMin = nRangeMin - nTolerance;
	DINT nMax = nRangeMax + nTolerance;
	if(nValue >= nMin && nValue <= nMax)
	{
		bResult = 1;
	}
	return bResult;
}

// NOLINTEND(readability-*, bugprone-easily-swappable-parameters, clang-diagnostic-invalid-utf8, clang-diagnostic-invalid-source-encoding, clang-diagnostic-pointer-arith, clang-diagnostic-strict-prototypes, hicpp-uppercase-literal-suffix, cppcoreguidelines-*, performance-*)
```
